// TwinCAT 3 PLC project Modbus
// ProgramVersion: 3.1.4022.7
// libraries:
//   LCLS Vacuum, * (SLAC - LCLS)
//   Tc2_ModbusRTU, * (Beckhoff Automation GmbH)
//   Tc2_ModbusSrv, * (Beckhoff Automation GmbH)
//   Tc2_Standard, * (Beckhoff Automation GmbH)
//   Tc2_System, * (Beckhoff Automation GmbH)
//   Tc3_Module, * (Beckhoff Automation GmbH)
// project tree:
//   / PlcTask.TcTTO
//   POUs/ FB_GaugeModbus.TcPOU, MAIN.TcPOU
//   POUs/Modbus/ p_ModbusRx_OutputCoils.TcPOU, p_ModbusRx_OutputReg.TcPOU, p_ModbusRx_PLCMemory.TcPOU, p_ModbusTx_InputCoils.TcPOU, p_ModbusTx_InputReg.TcPOU, p_ModbusTx_OutputCoils.TcPOU, p_ModbusTx_OutputReg.TcPOU, p_ModbusTx_PLCMemory.TcPOU, p_XLegacyPLCModbus.TcPOU
// real-time tasks:
//   TASK PlcTask: cycle T#10ms, priority 20, ADS port 350

CONFIGURATION Modbus
    RESOURCE PLC ON TwinCAT3
        TASK PlcTask(INTERVAL := T#10ms, PRIORITY := 20);
        PROGRAM MAIN WITH PlcTask : MAIN;
    END_RESOURCE
END_CONFIGURATION

// ---- POUs/MAIN.TcPOU
PROGRAM MAIN
VAR
	test:FB_GaugeModbus;
	
END_VAR

test(IP:='172.21.84.44',nMBAddr:=2048(*8#4000*),iBitOffset:=24);

END_PROGRAM

// ---- POUs/FB_GaugeModbus.TcPOU
FUNCTION_BLOCK FB_GaugeModbus EXTENDS FB_GaugeBase
VAR_INPUT
	IP: STRING;	//IP of Legacy PLC
    nMBAddr	:WORD; //Start address of the Register Memory
	iBitOffset:INT :=24;
	tTimeout :TIME:= T#5s;
END_VAR
VAR_OUTPUT
	VG: ST_VG;
	xNoPLCResponse: BOOL;
END_VAR
VAR
	fbPLCInputCoilsRx	:	FB_MBReadInputs;// (Modbus function 2)
	i_PLC_nBits	:	ARRAY [1..4] OF BYTE;
	ftReset	: F_TRIG; 
	tonRetry : TON;
	ErrCount:INT :=0;
END_VAR

A_ReadMB();

ACTION A_ReadMB:
(*Credit to Alex Wallace*)
(* Modbus Info for Koyo
Modbus Addresses for
Koyo DL05/06/240/250/260/430/440/450 PLCs
PLC Memory Type		| Modbus start address Decimal (octal) | Function codes
Inputs (X)			  2048 (04000)							2
Special Relays (SP)	  3072 (06000)							2
Outputs (Y)			  2048 (04000)							1, 5, 15
Control Relays (C)	  3072 (06000)							1, 5, 15
Timer Contacts (T)	  6144 (014000)							1, 5, 15
Counter Contacts (CT) 6400 (014400)							1, 5, 15
Stage Status Bits (S) 6144 (012000)							1, 5, 15
*)

// Retry after some time
tonRetry.IN := NOT fbPLCInputCoilsRx.bBusy;
tonRetry.PT := T#10S;
tonRetry();

ftReset(CLK:=fbPLCInputCoilsRx.bBusy);
fbPLCInputCoilsRx.bExecute := ftReset.Q OR tonRetry.Q;

fbPLCInputCoilsRx(sIPAddr:=IP, nTCPPort:=502, nQuantity:=24, nMBAddr:=nMBAddr(*+INT_TO_WORD(iBitOffset)*), cbLength:=SIZEOF(i_PLC_nBits),  pDestAddr:=ADR(i_PLC_nBits), tTimeout:=tTimeout);
//if there's a modbus error, set all incoming bits to zero
IF fbPLCInputCoilsRx.bError THEN
	i_PLC_nBits[1].0 := 0;
	i_PLC_nBits[1].1 := 0;
	i_PLC_nBits[1].2 := 0;
	i_PLC_nBits[1].3 := 0;
	i_PLC_nBits[1].4 := 0;
	i_PLC_nBits[1].5 := 0;
	i_PLC_nBits[1].6 := 0;
	i_PLC_nBits[1].7 := 0;
	i_PLC_nBits[2].0 := 0;
	i_PLC_nBits[2].1 := 0;
	i_PLC_nBits[2].2 := 0;
	i_PLC_nBits[2].3 := 0;
	i_PLC_nBits[2].4 := 0;
	i_PLC_nBits[2].5 := 0;
	i_PLC_nBits[2].6 := 0;
	i_PLC_nBits[2].7 := 0;
	VG.xPRESS_OK := FALSE;
	xNoPLCResponse:= TRUE;	
ELSIF NOT ftReset.Q AND fbPLCInputCoilsRx.cbRead > 0 THEN
	xNoPLCResponse:= FALSE;
	VG.rPRESS := 1E-8;
	VG.xPRESS_OK := i_PLC_nBits[0].0;
	fbPLCInputCoilsRx.bExecute :=False;
ELSIF (*ftReset.Q*) NOT (fbPLCInputCoilsRx.bExecute) AND fbPLCInputCoilsRx.cbRead = 0 THEN
	xNoPLCResponse:= TRUE;		
END_IF

// Log Action
tAction(CLK:=   fbPLCInputCoilsRx.bError or xNoPLCResponse);
IF tAction.Q THEN 
ErrCount:= ErrCount+1; 
fbLogger(sMsg:='Modbus read error', eSevr:=TcEventSeverity.Critical);
END_IF
END_ACTION

END_FUNCTION_BLOCK

// ---- POUs/Modbus/p_ModbusRx_OutputCoils.TcPOU
PROGRAM p_ModbusRx_OutputCoils
VAR
END_VAR

//mb_Output_Coils[0];  //System Controls
g_stSystem.xOverrideMode:=mb_Output_Coils[1];  //System Controls
//mb_Output_Coils[2];  //System Controls
//mb_Output_Coils[3];  //System Controls
//mb_Output_Coils[4];  //System Controls
//mb_Output_Coils[5];  //System Controls
//mb_Output_Coils[6];  //System Controls
//mb_Output_Coils[7];  //System Controls
//mb_Output_Coils[8];  //System Controls
//mb_Output_Coils[9];  //System Controls
vgcPBT_VGC_01.xOPN_SW:=mb_Output_Coils[10];  //Valve switch controls
vgcPBT_VGC_02.xOPN_SW:=mb_Output_Coils[11];  //Valve switch controls
vgcPBT_VGC_03.xOPN_SW:=mb_Output_Coils[12];  //Valve switch controls
vgcPBT_VGC_04.xOPN_SW:=mb_Output_Coils[13];  //Valve switch controls
//mb_Output_Coils[14];  //Valve switch controls
//mb_Output_Coils[15];  //Valve switch controls
//mb_Output_Coils[16];  //Valve switch controls
//mb_Output_Coils[17];  //Valve switch controls
//mb_Output_Coils[18];  //Valve switch controls
//mb_Output_Coils[19];  //Valve switch controls
//mb_Output_Coils[20];  //Valve switch controls
//mb_Output_Coils[21];  //Valve switch controls
//mb_Output_Coils[22];  //Valve switch controls
//mb_Output_Coils[23];  //Valve switch controls
//mb_Output_Coils[24];  //Valve switch controls
//mb_Output_Coils[25];  //Valve switch controls
//mb_Output_Coils[26];  //Valve switch controls
//mb_Output_Coils[27];  //Valve switch controls
//mb_Output_Coils[28];  //Valve switch controls
//mb_Output_Coils[29];  //Valve switch controls
//mb_Output_Coils[30];  //Valve switch controls
//mb_Output_Coils[31];  //Valve switch controls
//mb_Output_Coils[32];  //Valve switch controls
//mb_Output_Coils[33];  //Valve switch controls
//mb_Output_Coils[34];  //Valve switch controls
//mb_Output_Coils[35];  //Valve switch controls
//mb_Output_Coils[36];  //Valve switch controls
//mb_Output_Coils[37];  //Valve switch controls
//mb_Output_Coils[38];  //Valve switch controls
//mb_Output_Coils[39];  //Valve switch controls
//mb_Output_Coils[40];  //Valve switch controls
//mb_Output_Coils[41];  //Valve switch controls
//mb_Output_Coils[42];  //Valve switch controls
//mb_Output_Coils[43];  //Valve switch controls
//mb_Output_Coils[44];  //Valve switch controls
//mb_Output_Coils[45];  //Valve switch controls
//mb_Output_Coils[46];  //Valve switch controls
//mb_Output_Coils[47];  //Valve switch controls
//mb_Output_Coils[48];  //Valve switch controls
//mb_Output_Coils[49];  //Valve switch controls
//mb_Output_Coils[50];  //Valve switch controls
//mb_Output_Coils[51];  //Valve switch controls
//mb_Output_Coils[52];  //Valve switch controls
//mb_Output_Coils[53];  //Valve switch controls
//mb_Output_Coils[54];  //Valve switch controls
//mb_Output_Coils[55];  //Valve switch controls
//mb_Output_Coils[56];  //Valve switch controls
//mb_Output_Coils[57];  //Valve switch controls
//mb_Output_Coils[58];  //Valve switch controls
//mb_Output_Coils[59];  //Valve switch controls
//mb_Output_Coils[60];  //Valve switch controls
//mb_Output_Coils[61];  //Valve switch controls
//mb_Output_Coils[62];  //Valve switch controls
//mb_Output_Coils[63];  //Valve switch controls
//mb_Output_Coils[64];  //Valve switch controls
//mb_Output_Coils[65];  //Valve switch controls
//mb_Output_Coils[66];  //Valve switch controls
//mb_Output_Coils[67];  //Valve switch controls
//mb_Output_Coils[68];  //Valve switch controls
//mb_Output_Coils[69];  //Valve switch controls
//mb_Output_Coils[70];  //Turbo Controls
//mb_Output_Coils[71];  //Turbo Controls
//mb_Output_Coils[72];  //Turbo Controls
//mb_Output_Coils[74];  //Turbo Controls
//mb_Output_Coils[75];  //Turbo Controls
//mb_Output_Coils[76];  //Turbo Controls
//mb_Output_Coils[77];  //Turbo Controls
//mb_Output_Coils[78];  //Turbo Controls
//mb_Output_Coils[79];  //Turbo Controls
//mb_Output_Coils[80];  //Turbo Controls
//mb_Output_Coils[81];  //Turbo Controls
//mb_Output_Coils[82];  //Turbo Controls
//mb_Output_Coils[83];  //Turbo Controls
//mb_Output_Coils[84];  //Turbo Controls
//mb_Output_Coils[85];  //Turbo Controls
//mb_Output_Coils[86];  //Turbo Controls
//mb_Output_Coils[87];  //Turbo Controls
//mb_Output_Coils[88];  //Turbo Controls
//mb_Output_Coils[89];  //Turbo Controls
//mb_Output_Coils[90];  //Turbo Controls
//mb_Output_Coils[91];  //Turbo Controls
//mb_Output_Coils[92];  //Turbo Controls
//mb_Output_Coils[93];  //Turbo Controls
//mb_Output_Coils[94];  //Turbo Controls
//mb_Output_Coils[95];  //Turbo Controls
//mb_Output_Coils[96];  //Turbo Controls
//mb_Output_Coils[97];  //Turbo Controls
//mb_Output_Coils[98];  //Turbo Controls
//mb_Output_Coils[99];  //Turbo Controls
//mb_Output_Coils[100];  //Turbo Controls
//mb_Output_Coils[101];  //Turbo Controls
//mb_Output_Coils[102];  //Turbo Controls
//mb_Output_Coils[103];  //Turbo Controls
//mb_Output_Coils[104];  //Turbo Controls
//mb_Output_Coils[105];  //Turbo Controls
//mb_Output_Coils[106];  //Turbo Controls
//mb_Output_Coils[107];  //Turbo Controls
//mb_Output_Coils[108];  //Turbo Controls
//mb_Output_Coils[109];  //Turbo Controls
//mb_Output_Coils[110];  //Turbo Controls
//mb_Output_Coils[111];  //Turbo Controls
//mb_Output_Coils[112];  //Turbo Controls
//mb_Output_Coils[113];  //Turbo Controls
//mb_Output_Coils[114];  //Turbo Controls
//mb_Output_Coils[115];  //Turbo Controls
//mb_Output_Coils[116];  //Turbo Controls
//mb_Output_Coils[117];  //Turbo Controls
//mb_Output_Coils[118];  //Turbo Controls
//mb_Output_Coils[119];  //Turbo Controls
vgPBT_GCC_02.xHV_SW:=mb_Output_Coils[120];  //CC HV Enable
vgPBT_GCC_04.xHV_SW:=mb_Output_Coils[121];  //CC HV Enable
vgPBT_GCC_06.xHV_SW:=mb_Output_Coils[122];  //CC HV Enable
vgPBT_GCC_07.xHV_SW:=mb_Output_Coils[123];  //CC HV Enable
vgPBT_GCC_09.xHV_SW:=mb_Output_Coils[124];  //CC HV Enable
//mb_Output_Coils[125];  //CC HV Enable
//mb_Output_Coils[126];  //CC HV Enable
//mb_Output_Coils[127];  //CC HV Enable
//mb_Output_Coils[128];  //CC HV Enable
//mb_Output_Coils[129];  //CC HV Enable
//mb_Output_Coils[130];  //CC HV Enable
//mb_Output_Coils[131];  //CC HV Enable
//mb_Output_Coils[132];  //CC HV Enable
//mb_Output_Coils[133];  //CC HV Enable
//mb_Output_Coils[134];  //CC HV Enable
//mb_Output_Coils[135];  //CC HV Enable
//mb_Output_Coils[136];  //CC HV Enable
//mb_Output_Coils[137];  //CC HV Enable
//mb_Output_Coils[138];  //CC HV Enable
//mb_Output_Coils[139];  //CC HV Enable
//mb_Output_Coils[140];  //CC HV Enable
//mb_Output_Coils[141];  //CC HV Enable
//mb_Output_Coils[142];  //CC HV Enable
//mb_Output_Coils[143];  //CC HV Enable
//mb_Output_Coils[144];  //CC HV Enable
//mb_Output_Coils[145];  //CC HV Enable
//mb_Output_Coils[146];  //CC HV Enable
//mb_Output_Coils[147];  //CC HV Enable
//mb_Output_Coils[148];  //CC HV Enable
//mb_Output_Coils[149];  //CC HV Enable
//mb_Output_Coils[150];  //CC HV Enable
//mb_Output_Coils[151];  //CC HV Enable
//mb_Output_Coils[152];  //CC HV Enable
//mb_Output_Coils[153];  //CC HV Enable
//mb_Output_Coils[154];  //CC HV Enable
//mb_Output_Coils[155];  //CC HV Enable
//mb_Output_Coils[156];  //CC HV Enable
//mb_Output_Coils[157];  //CC HV Enable
//mb_Output_Coils[158];  //CC HV Enable
//mb_Output_Coils[159];  //CC HV Enable
//mb_Output_Coils[160];  //
//mb_Output_Coils[161];  //
//mb_Output_Coils[162];  //
//mb_Output_Coils[163];  //
//mb_Output_Coils[164];  //
//mb_Output_Coils[165];  //
//mb_Output_Coils[166];  //
//mb_Output_Coils[167];  //
//mb_Output_Coils[168];  //
//mb_Output_Coils[169];  //
//mb_Output_Coils[170];  //
//mb_Output_Coils[171];  //
//mb_Output_Coils[172];  //
//mb_Output_Coils[173];  //
//mb_Output_Coils[174];  //
//mb_Output_Coils[175];  //
//mb_Output_Coils[176];  //
//mb_Output_Coils[177];  //
//mb_Output_Coils[178];  //
//mb_Output_Coils[179];  //
//mb_Output_Coils[180];  //
//mb_Output_Coils[181];  //
//mb_Output_Coils[182];  //
//mb_Output_Coils[183];  //
//mb_Output_Coils[184];  //
//mb_Output_Coils[185];  //
//mb_Output_Coils[186];  //
//mb_Output_Coils[187];  //
//mb_Output_Coils[188];  //
//mb_Output_Coils[189];  //
//mb_Output_Coils[190];  //
//mb_Output_Coils[191];  //
//mb_Output_Coils[192];  //
//mb_Output_Coils[193];  //
//mb_Output_Coils[194];  //
//mb_Output_Coils[195];  //
//mb_Output_Coils[196];  //
//mb_Output_Coils[197];  //
//mb_Output_Coils[198];  //
//mb_Output_Coils[199];  //
vgcPBT_VGC_01.xOvrdOpn:=mb_Output_Coils[200];  //Valve overrides
vgcPBT_VGC_02.xOvrdOpn:=mb_Output_Coils[201];  //Valve overrides
vgcPBT_VGC_03.xOvrdOpn:=mb_Output_Coils[202];  //Valve overrides
vgcPBT_VGC_04.xOvrdOpn:=mb_Output_Coils[203];  //Valve overrides
//mb_Output_Coils[204];  //
//mb_Output_Coils[205];  //
//mb_Output_Coils[206];  //
//mb_Output_Coils[207];  //
//mb_Output_Coils[208];  //
//mb_Output_Coils[209];  //
//mb_Output_Coils[210];  //
//mb_Output_Coils[211];  //
//mb_Output_Coils[212];  //
//mb_Output_Coils[213];  //
//mb_Output_Coils[214];  //
//mb_Output_Coils[215];  //
//mb_Output_Coils[216];  //
//mb_Output_Coils[217];  //
//mb_Output_Coils[218];  //
//mb_Output_Coils[219];  //
//mb_Output_Coils[220];  //
//mb_Output_Coils[221];  //
//mb_Output_Coils[222];  //
//mb_Output_Coils[223];  //
//mb_Output_Coils[224];  //
//mb_Output_Coils[225];  //
//mb_Output_Coils[226];  //
//mb_Output_Coils[227];  //
//mb_Output_Coils[228];  //
//mb_Output_Coils[229];  //
//mb_Output_Coils[230];  //
//mb_Output_Coils[231];  //
//mb_Output_Coils[232];  //
//mb_Output_Coils[233];  //
//mb_Output_Coils[234];  //
//mb_Output_Coils[235];  //
//mb_Output_Coils[236];  //
//mb_Output_Coils[237];  //
//mb_Output_Coils[238];  //
//mb_Output_Coils[239];  //
//mb_Output_Coils[240];  //
//mb_Output_Coils[241];  //
//mb_Output_Coils[242];  //
//mb_Output_Coils[243];  //
//mb_Output_Coils[244];  //
//mb_Output_Coils[245];  //
//mb_Output_Coils[246];  //
//mb_Output_Coils[247];  //
//mb_Output_Coils[248];  //
//mb_Output_Coils[249];  //
//mb_Output_Coils[250];  //
//mb_Output_Coils[251];  //
//mb_Output_Coils[252];  //
//mb_Output_Coils[253];  //
//mb_Output_Coils[254];  //
//mb_Output_Coils[255];  //

END_PROGRAM

// ---- POUs/Modbus/p_ModbusRx_OutputReg.TcPOU
PROGRAM p_ModbusRx_OutputReg
VAR
END_VAR

//mb_Output_Registers[0];  //System parameters
//mb_Output_Registers[1];  //System parameters
//mb_Output_Registers[2];  //System parameters
//mb_Output_Registers[3];  //System parameters
//mb_Output_Registers[4];  //System parameters
//mb_Output_Registers[5];  //System parameters
//mb_Output_Registers[6];  //System parameters
//mb_Output_Registers[7];  //System parameters
//mb_Output_Registers[8];  //System parameters
//mb_Output_Registers[9];  //System parameters
//mb_Output_Registers[10];  //VG setpoint
//mb_Output_Registers[11];  //VG setpoint
//mb_Output_Registers[12];  //VG setpoint
//mb_Output_Registers[13];  //VG setpoint
//mb_Output_Registers[14];  //VG setpoint
//mb_Output_Registers[15];  //VG setpoint
//mb_Output_Registers[16];  //VG setpoint
//mb_Output_Registers[17];  //VG setpoint
//mb_Output_Registers[18];  //VG setpoint
//mb_Output_Registers[19];  //VG setpoint
//mb_Output_Registers[20];  //VG setpoint
//mb_Output_Registers[21];  //VG setpoint
//mb_Output_Registers[22];  //VG setpoint
//mb_Output_Registers[23];  //VG setpoint
//mb_Output_Registers[24];  //VG setpoint
//mb_Output_Registers[25];  //VG setpoint
//mb_Output_Registers[26];  //VG setpoint
//mb_Output_Registers[27];  //VG setpoint
//mb_Output_Registers[28];  //VG setpoint
//mb_Output_Registers[29];  //VG setpoint
//mb_Output_Registers[30];  //VG setpoint
//mb_Output_Registers[31];  //VG setpoint
//mb_Output_Registers[32];  //VG setpoint
//mb_Output_Registers[33];  //VG setpoint
//mb_Output_Registers[34];  //VG setpoint
//mb_Output_Registers[35];  //VG setpoint
//mb_Output_Registers[36];  //VG setpoint
//mb_Output_Registers[37];  //VG setpoint
//mb_Output_Registers[38];  //VG setpoint
//mb_Output_Registers[39];  //VG setpoint
//mb_Output_Registers[40];  //VG setpoint
//mb_Output_Registers[41];  //VG setpoint
//mb_Output_Registers[42];  //VG setpoint
//mb_Output_Registers[43];  //VG setpoint
//mb_Output_Registers[44];  //VG setpoint
//mb_Output_Registers[45];  //VG setpoint
//mb_Output_Registers[46];  //VG setpoint
//mb_Output_Registers[47];  //VG setpoint
//mb_Output_Registers[48];  //VG setpoint
//mb_Output_Registers[49];  //VG setpoint
//mb_Output_Registers[50];  //VG setpoint
//mb_Output_Registers[51];  //VG setpoint
//mb_Output_Registers[52];  //VG setpoint
//mb_Output_Registers[53];  //VG setpoint
//mb_Output_Registers[54];  //VG setpoint
//mb_Output_Registers[55];  //VG setpoint
//mb_Output_Registers[56];  //VG setpoint
//mb_Output_Registers[57];  //VG setpoint
//mb_Output_Registers[58];  //VG setpoint
//mb_Output_Registers[59];  //VG setpoint
//mb_Output_Registers[60];  //default
//mb_Output_Registers[61];  //default
//mb_Output_Registers[62];  //default
//mb_Output_Registers[63];  //default
//mb_Output_Registers[64];  //default
//mb_Output_Registers[65];  //default
//mb_Output_Registers[66];  //default
//mb_Output_Registers[67];  //default
//mb_Output_Registers[68];  //default
//mb_Output_Registers[69];  //default
//mb_Output_Registers[70];  //default
//mb_Output_Registers[71];  //default
//mb_Output_Registers[72];  //default
//mb_Output_Registers[73];  //default
//mb_Output_Registers[74];  //default
//mb_Output_Registers[75];  //default
//mb_Output_Registers[76];  //default
//mb_Output_Registers[77];  //default
//mb_Output_Registers[78];  //default
//mb_Output_Registers[79];  //default
//mb_Output_Registers[80];  //default
//mb_Output_Registers[81];  //default
//mb_Output_Registers[82];  //default
//mb_Output_Registers[83];  //default
//mb_Output_Registers[84];  //default
//mb_Output_Registers[85];  //default
//mb_Output_Registers[86];  //default
//mb_Output_Registers[87];  //default
//mb_Output_Registers[88];  //default
//mb_Output_Registers[89];  //default
//mb_Output_Registers[90];  //default
//mb_Output_Registers[91];  //default
//mb_Output_Registers[92];  //default
//mb_Output_Registers[93];  //default
//mb_Output_Registers[94];  //default
//mb_Output_Registers[95];  //default
//mb_Output_Registers[96];  //default
//mb_Output_Registers[97];  //default
//mb_Output_Registers[98];  //default
//mb_Output_Registers[99];  //default
//mb_Output_Registers[100];  //default
//mb_Output_Registers[101];  //default
//mb_Output_Registers[102];  //default
//mb_Output_Registers[103];  //default
//mb_Output_Registers[104];  //default
//mb_Output_Registers[105];  //default
//mb_Output_Registers[106];  //default
//mb_Output_Registers[107];  //default
//mb_Output_Registers[108];  //default
//mb_Output_Registers[109];  //default
//mb_Output_Registers[110];  //default
//mb_Output_Registers[111];  //default
//mb_Output_Registers[112];  //default
//mb_Output_Registers[113];  //default
//mb_Output_Registers[114];  //default
//mb_Output_Registers[115];  //default
//mb_Output_Registers[116];  //default
//mb_Output_Registers[117];  //default
//mb_Output_Registers[118];  //default
//mb_Output_Registers[119];  //default
//mb_Output_Registers[120];  //default
//mb_Output_Registers[121];  //default
//mb_Output_Registers[122];  //default
//mb_Output_Registers[123];  //default
//mb_Output_Registers[124];  //default
//mb_Output_Registers[125];  //default
//mb_Output_Registers[126];  //default
//mb_Output_Registers[127];  //default
//mb_Output_Registers[128];  //default
//mb_Output_Registers[129];  //default
//mb_Output_Registers[130];  //default
//mb_Output_Registers[131];  //default
//mb_Output_Registers[132];  //default
//mb_Output_Registers[133];  //default
//mb_Output_Registers[134];  //default
//mb_Output_Registers[135];  //default
//mb_Output_Registers[136];  //default
//mb_Output_Registers[137];  //default
//mb_Output_Registers[138];  //default
//mb_Output_Registers[139];  //default
//mb_Output_Registers[140];  //default
//mb_Output_Registers[141];  //default
//mb_Output_Registers[142];  //default
//mb_Output_Registers[143];  //default
//mb_Output_Registers[144];  //default
//mb_Output_Registers[145];  //default
//mb_Output_Registers[146];  //default
//mb_Output_Registers[147];  //default
//mb_Output_Registers[148];  //default
//mb_Output_Registers[149];  //default
//mb_Output_Registers[150];  //default
//mb_Output_Registers[151];  //default
//mb_Output_Registers[152];  //default
//mb_Output_Registers[153];  //default
//mb_Output_Registers[154];  //default
//mb_Output_Registers[155];  //default
//mb_Output_Registers[156];  //default
//mb_Output_Registers[157];  //default
//mb_Output_Registers[158];  //default
//mb_Output_Registers[159];  //default
//mb_Output_Registers[160];  //default
//mb_Output_Registers[161];  //default
//mb_Output_Registers[162];  //default
//mb_Output_Registers[163];  //default
//mb_Output_Registers[164];  //default
//mb_Output_Registers[165];  //default
//mb_Output_Registers[166];  //default
//mb_Output_Registers[167];  //default
//mb_Output_Registers[168];  //default
//mb_Output_Registers[169];  //default
//mb_Output_Registers[170];  //default
//mb_Output_Registers[171];  //default
//mb_Output_Registers[172];  //default
//mb_Output_Registers[173];  //default
//mb_Output_Registers[174];  //default
//mb_Output_Registers[175];  //default
//mb_Output_Registers[176];  //default
//mb_Output_Registers[177];  //default
//mb_Output_Registers[178];  //default
//mb_Output_Registers[179];  //default
//mb_Output_Registers[180];  //default
//mb_Output_Registers[181];  //default
//mb_Output_Registers[182];  //default
//mb_Output_Registers[183];  //default
//mb_Output_Registers[184];  //default
//mb_Output_Registers[185];  //default
//mb_Output_Registers[186];  //default
//mb_Output_Registers[187];  //default
//mb_Output_Registers[188];  //default
//mb_Output_Registers[189];  //default
//mb_Output_Registers[190];  //default
//mb_Output_Registers[191];  //default
//mb_Output_Registers[192];  //default
//mb_Output_Registers[193];  //default
//mb_Output_Registers[194];  //default
//mb_Output_Registers[195];  //default
//mb_Output_Registers[196];  //default
//mb_Output_Registers[197];  //default
//mb_Output_Registers[198];  //default
//mb_Output_Registers[199];  //default
//mb_Output_Registers[200];  //default
//mb_Output_Registers[201];  //default
//mb_Output_Registers[202];  //default
//mb_Output_Registers[203];  //default
//mb_Output_Registers[204];  //default
//mb_Output_Registers[205];  //default
//mb_Output_Registers[206];  //default
//mb_Output_Registers[207];  //default
//mb_Output_Registers[208];  //default
//mb_Output_Registers[209];  //default
//mb_Output_Registers[210];  //default
//mb_Output_Registers[211];  //default
//mb_Output_Registers[212];  //default
//mb_Output_Registers[213];  //default
//mb_Output_Registers[214];  //default
//mb_Output_Registers[215];  //default
//mb_Output_Registers[216];  //default
//mb_Output_Registers[217];  //default
//mb_Output_Registers[218];  //default
//mb_Output_Registers[219];  //default
//mb_Output_Registers[220];  //default
//mb_Output_Registers[221];  //default
//mb_Output_Registers[222];  //default
//mb_Output_Registers[223];  //default
//mb_Output_Registers[224];  //default
//mb_Output_Registers[225];  //default
//mb_Output_Registers[226];  //default
//mb_Output_Registers[227];  //default
//mb_Output_Registers[228];  //default
//mb_Output_Registers[229];  //default
//mb_Output_Registers[230];  //default
//mb_Output_Registers[231];  //default
//mb_Output_Registers[232];  //default
//mb_Output_Registers[233];  //default
//mb_Output_Registers[234];  //default
//mb_Output_Registers[235];  //default
//mb_Output_Registers[236];  //default
//mb_Output_Registers[237];  //default
//mb_Output_Registers[238];  //default
//mb_Output_Registers[239];  //default
//mb_Output_Registers[240];  //default
//mb_Output_Registers[241];  //default
//mb_Output_Registers[242];  //default
//mb_Output_Registers[243];  //default
//mb_Output_Registers[244];  //default
//mb_Output_Registers[245];  //default
//mb_Output_Registers[246];  //default
//mb_Output_Registers[247];  //default
//mb_Output_Registers[248];  //default
//mb_Output_Registers[249];  //default
//mb_Output_Registers[250];  //default
//mb_Output_Registers[251];  //default
//mb_Output_Registers[252];  //default
//mb_Output_Registers[253];  //default
//mb_Output_Registers[254];  //default
//mb_Output_Registers[255];  //default

END_PROGRAM

// ---- POUs/Modbus/p_ModbusRx_PLCMemory.TcPOU
PROGRAM p_ModbusRx_PLCMemory
VAR
END_VAR

MEMCPY(destAddr:=ADR(mb_PLC_Memory[70]), srcAddr:=ADR(vgPBT_GCC_02.rVAC_SP), n:=SIZEOF(vgPBT_GCC_02.rVAC_SP));  //VG pressure sp readbacks
MEMCPY(destAddr:=ADR(mb_PLC_Memory[72]), srcAddr:=ADR(vgPBT_GPI_02.rVAC_SP), n:=SIZEOF(vgPBT_GPI_02.rVAC_SP));  //VG pressure sp readbacks

MEMCPY(destAddr:=ADR(mb_PLC_Memory[74]), srcAddr:=ADR(vgPBT_GCC_04.rVAC_SP), n:=SIZEOF(vgPBT_GCC_04.rVAC_SP));  //VG pressure sp readbacks
MEMCPY(destAddr:=ADR(mb_PLC_Memory[76]), srcAddr:=ADR(vgPBT_GPI_04.rVAC_SP), n:=SIZEOF(vgPBT_GPI_04.rVAC_SP));  //VG pressure sp readbacks

MEMCPY(destAddr:=ADR(mb_PLC_Memory[78]), srcAddr:=ADR(vgPBT_GCC_06.rVAC_SP), n:=SIZEOF(vgPBT_GCC_06.rVAC_SP));  //VG pressure sp readbacks
MEMCPY(destAddr:=ADR(mb_PLC_Memory[80]), srcAddr:=ADR(vgPBT_GPI_06.rVAC_SP), n:=SIZEOF(vgPBT_GPI_06.rVAC_SP));  //VG pressure sp readbacks

MEMCPY(destAddr:=ADR(mb_PLC_Memory[82]), srcAddr:=ADR(vgPBT_GCC_07.rVAC_SP), n:=SIZEOF(vgPBT_GCC_07.rVAC_SP));  //VG pressure sp readbacks
MEMCPY(destAddr:=ADR(mb_PLC_Memory[84]), srcAddr:=ADR(vgPBT_GPI_07.rVAC_SP), n:=SIZEOF(vgPBT_GPI_07.rVAC_SP));  //VG pressure sp readbacks

MEMCPY(destAddr:=ADR(mb_PLC_Memory[86]), srcAddr:=ADR(vgPBT_GCC_09.rVAC_SP), n:=SIZEOF(vgPBT_GCC_09.rVAC_SP));  //VG pressure sp readbacks
MEMCPY(destAddr:=ADR(mb_PLC_Memory[88]), srcAddr:=ADR(vgPBT_GPI_09.rVAC_SP), n:=SIZEOF(vgPBT_GPI_09.rVAC_SP));  //VG pressure sp readbacks

END_PROGRAM

// ---- POUs/Modbus/p_ModbusTx_InputCoils.TcPOU
PROGRAM p_ModbusTx_InputCoils
VAR
	
END_VAR

VAR_OUTPUT
	

	XHV_DIS: BOOL;
END_VAR

mb_Input_Coils[0]:=FALSE;  //default
//mb_Input_Coils[1]:=i_xMFX_ppsStopperPos_Out;  //default
//mb_Input_Coils[2]:=i_xMFX_ppsStopperPos_In;  //default
mb_Input_Coils[3]:=q_xXCS_MPSOK;  //default
mb_Input_Coils[4]:=g_xIOState;  //default
//mb_Input_Coils[5]:=i_xDG1_MMS01_OUT;  //default
mb_Input_Coils[6]:=FALSE;  //default
mb_Input_Coils[7]:=FALSE;  //default
mb_Input_Coils[8]:=FALSE;  //default
mb_Input_Coils[9]:=FALSE;  //default
mb_Input_Coils[10]:=vgcPBT_VGC_01.i_xOpnLS;  //Valve position readbacks
mb_Input_Coils[11]:=vgcPBT_VGC_01.i_xClsLS;  //Valve position readbacks
mb_Input_Coils[12]:=vgcPBT_VGC_02.i_xOpnLS;  //Valve position readbacks
mb_Input_Coils[13]:=vgcPBT_VGC_02.i_xClsLS;  //Valve position readbacks
mb_Input_Coils[14]:=vgcPBT_VGC_03.i_xOpnLS;  //Valve position readbacks
mb_Input_Coils[15]:=vgcPBT_VGC_03.i_xClsLS;  //Valve position readbacks
mb_Input_Coils[16]:=vgcPBT_VGC_04.i_xOpnLS;  //Valve position readbacks
mb_Input_Coils[17]:=vgcPBT_VGC_04.i_xClsLS;  //Valve position readbacks
mb_Input_Coils[18]:=FALSE;  //Valve position readbacks
mb_Input_Coils[19]:=FALSE;  //Valve position readbacks
mb_Input_Coils[20]:=FALSE; //Valve position readbacks
mb_Input_Coils[21]:=FALSE;  //Valve position readbacks
mb_Input_Coils[22]:=FALSE;  //Valve position readbacks
mb_Input_Coils[23]:=FALSE;  //Valve position readbacks
mb_Input_Coils[24]:=FALSE;  //Valve position readbacks
mb_Input_Coils[25]:=FALSE;  //Valve position readbacks
mb_Input_Coils[26]:=FALSE;  //Valve position readbacks
mb_Input_Coils[27]:=FALSE;  //Valve position readbacks
mb_Input_Coils[28]:=FALSE;  //Valve position readbacks
mb_Input_Coils[29]:=FALSE;  //Valve position readbacks
mb_Input_Coils[30]:=FALSE;  //Valve position readbacks
mb_Input_Coils[31]:=FALSE;  //Valve position readbacks
mb_Input_Coils[32]:=FALSE;  //Valve position readbacks
mb_Input_Coils[33]:=FALSE;  //Valve position readbacks
mb_Input_Coils[34]:=FALSE;  //Valve position readbacks
mb_Input_Coils[35]:=FALSE;  //Valve position readbacks
mb_Input_Coils[36]:=FALSE;  //Valve position readbacks
mb_Input_Coils[37]:=FALSE;  //Valve position readbacks
mb_Input_Coils[38]:=FALSE;  //Valve position readbacks
mb_Input_Coils[39]:=FALSE;  //Valve position readbacks
mb_Input_Coils[40]:=FALSE;  //Valve position readbacks
mb_Input_Coils[41]:=FALSE;  //Valve position readbacks
mb_Input_Coils[42]:=FALSE;  //Valve position readbacks
mb_Input_Coils[43]:=FALSE;  //Valve position readbacks
mb_Input_Coils[44]:=FALSE;  //Valve position readbacks
mb_Input_Coils[45]:=FALSE;  //Valve position readbacks
mb_Input_Coils[46]:=FALSE;  //Valve position readbacks
mb_Input_Coils[47]:=FALSE;  //Valve position readbacks
mb_Input_Coils[48]:=FALSE;  //Valve position readbacks
mb_Input_Coils[49]:=FALSE;  //Valve position readbacks
mb_Input_Coils[50]:=FALSE;  //Valve position readbacks
mb_Input_Coils[51]:=FALSE;  //Valve position readbacks
mb_Input_Coils[52]:=FALSE;  //Valve position readbacks
mb_Input_Coils[53]:=FALSE;  //Valve position readbacks
mb_Input_Coils[54]:=FALSE;  //Valve position readbacks
mb_Input_Coils[55]:=FALSE;  //Valve position readbacks
mb_Input_Coils[56]:=FALSE;  //Valve position readbacks
mb_Input_Coils[57]:=FALSE;  //Valve position readbacks
mb_Input_Coils[58]:=FALSE;  //Valve position readbacks
mb_Input_Coils[59]:=FALSE;  //Valve position readbacks
mb_Input_Coils[60]:=vgcPBT_VGC_01.xOPN_OK;  //Valve position readbacks
mb_Input_Coils[61]:=vgcPBT_VGC_02.xOPN_OK;  //Valve position readbacks
mb_Input_Coils[62]:=vgcPBT_VGC_03.xOPN_OK;  //Valve position readbacks
mb_Input_Coils[63]:=vgcPBT_VGC_04.xOPN_OK;  //Valve position readbacks
mb_Input_Coils[64]:=FALSE;  //Valve position readbacks
mb_Input_Coils[65]:=FALSE;  //Valve position readbacks
mb_Input_Coils[66]:=FALSE;  //Valve position readbacks
mb_Input_Coils[67]:=FALSE;  //Valve position readbacks
mb_Input_Coils[68]:=FALSE;  //Valve position readbacks
mb_Input_Coils[69]:=FALSE;  //Valve position readbacks
mb_Input_Coils[70]:=FALSE;  //Valve position readbacks
mb_Input_Coils[71]:=FALSE;  //Valve position readbacks
mb_Input_Coils[72]:=FALSE;  //Valve position readbacks
mb_Input_Coils[73]:=FALSE;  //Valve position readbacks
mb_Input_Coils[74]:=FALSE;  //Valve position readbacks
mb_Input_Coils[75]:=FALSE;  //Valve position readbacks
mb_Input_Coils[76]:=FALSE;  //Valve position readbacks
mb_Input_Coils[77]:=FALSE;  //Valve position readbacks
mb_Input_Coils[78]:=FALSE;  //Valve position readbacks
mb_Input_Coils[79]:=FALSE;  //Valve position readbacks
mb_Input_Coils[80]:=FALSE;  //Valve position readbacks
mb_Input_Coils[81]:=FALSE;  //Valve position readbacks
mb_Input_Coils[82]:=FALSE;  //Valve position readbacks
mb_Input_Coils[83]:=FALSE;  //Valve position readbacks
mb_Input_Coils[84]:=FALSE;  //Valve position readbacks
mb_Input_Coils[85]:=FALSE;  //Valve position readbacks
mb_Input_Coils[86]:=FALSE;  //Valve position readbacks
mb_Input_Coils[87]:=FALSE;  //Valve position readbacks
mb_Input_Coils[88]:=FALSE;  //Valve position readbacks
mb_Input_Coils[89]:=FALSE;  //Valve position readbacks
mb_Input_Coils[90]:=FALSE;  //Valve position readbacks
mb_Input_Coils[91]:=FALSE;  //Valve position readbacks
mb_Input_Coils[92]:=FALSE;  //Valve position readbacks
mb_Input_Coils[93]:=FALSE;  //Valve position readbacks
mb_Input_Coils[94]:=FALSE;  //Valve position readbacks
mb_Input_Coils[95]:=FALSE;  //Valve position readbacks
mb_Input_Coils[96]:=FALSE;  //Valve position readbacks
mb_Input_Coils[97]:=FALSE;  //Valve position readbacks
mb_Input_Coils[98]:=FALSE;  //Valve position readbacks
mb_Input_Coils[99]:=FALSE;  //Valve position readbacks
mb_Input_Coils[100]:=FALSE;  //Valve position readbacks
mb_Input_Coils[101]:=FALSE;  //Valve position readbacks
mb_Input_Coils[102]:=FALSE;  //Valve position readbacks
mb_Input_Coils[103]:=FALSE;  //Valve position readbacks
mb_Input_Coils[104]:=FALSE;  //Valve position readbacks
mb_Input_Coils[105]:=FALSE;  //Valve position readbacks
mb_Input_Coils[106]:=FALSE;  //Valve position readbacks
mb_Input_Coils[107]:=FALSE;  //Valve position readbacks
mb_Input_Coils[108]:=FALSE;  //Valve position readbacks
mb_Input_Coils[109]:=FALSE;  //Valve position readbacks
mb_Input_Coils[110]:=FALSE;  //Valve position readbacks
mb_Input_Coils[111]:=FALSE;  //Valve position readbacks
mb_Input_Coils[112]:=FALSE;  //Valve position readbacks
mb_Input_Coils[113]:=FALSE;  //Valve position readbacks
mb_Input_Coils[114]:=FALSE;  //Valve position readbacks
mb_Input_Coils[115]:=FALSE;  //Valve position readbacks
mb_Input_Coils[116]:=FALSE;  //Valve position readbacks
mb_Input_Coils[117]:=FALSE;  //Valve position readbacks
mb_Input_Coils[118]:=FALSE;  //Valve position readbacks
mb_Input_Coils[119]:=FALSE;  //Valve position readbacks
mb_Input_Coils[120]:=FALSE;  //Turbo pump readbacks
mb_Input_Coils[121]:=FALSE;  //Turbo pump readbacks
mb_Input_Coils[122]:=FALSE;  //Turbo pump readbacks
mb_Input_Coils[123]:=FALSE;  //Turbo pump readbacks
mb_Input_Coils[124]:=FALSE;  //Turbo pump readbacks
mb_Input_Coils[125]:=FALSE;  //Turbo pump readbacks
mb_Input_Coils[126]:=FALSE;  //Turbo pump readbacks
mb_Input_Coils[127]:=FALSE;  //Turbo pump readbacks
mb_Input_Coils[128]:=FALSE;  //Turbo pump readbacks
mb_Input_Coils[129]:=FALSE;  //Turbo pump readbacks
mb_Input_Coils[130]:=FALSE;  //Turbo pump readbacks
mb_Input_Coils[131]:=FALSE;  //Turbo pump readbacks
mb_Input_Coils[132]:=FALSE;  //Turbo pump readbacks
mb_Input_Coils[133]:=FALSE;  //Turbo pump readbacks
mb_Input_Coils[134]:=FALSE;  //Turbo pump readbacks
mb_Input_Coils[135]:=FALSE;  //Turbo pump readbacks
mb_Input_Coils[136]:=FALSE;  //Turbo pump readbacks
mb_Input_Coils[137]:=FALSE;  //Turbo pump readbacks
mb_Input_Coils[138]:=FALSE;  //Turbo pump readbacks
mb_Input_Coils[139]:=FALSE;  //Turbo pump readbacks
mb_Input_Coils[140]:=FALSE;  //Turbo pump readbacks
mb_Input_Coils[141]:=FALSE;  //Turbo pump readbacks
mb_Input_Coils[142]:=FALSE;  //Turbo pump readbacks
mb_Input_Coils[143]:=FALSE;  //Turbo pump readbacks
mb_Input_Coils[144]:=FALSE;  //Turbo pump readbacks
mb_Input_Coils[145]:=FALSE;  //Turbo pump readbacks
mb_Input_Coils[146]:=FALSE;  //Turbo pump readbacks
mb_Input_Coils[147]:=FALSE;  //Turbo pump readbacks
mb_Input_Coils[148]:=FALSE;  //Turbo pump readbacks
mb_Input_Coils[149]:=FALSE;  //Turbo pump readbacks
mb_Input_Coils[150]:=FALSE;  //Turbo pump readbacks
mb_Input_Coils[151]:=FALSE;  //Turbo pump readbacks
mb_Input_Coils[152]:=FALSE;  //Turbo pump readbacks
mb_Input_Coils[153]:=FALSE;  //Turbo pump readbacks
mb_Input_Coils[154]:=FALSE;  //Turbo pump readbacks
mb_Input_Coils[155]:=FALSE;  //Turbo pump readbacks
mb_Input_Coils[156]:=FALSE;  //Turbo pump readbacks
mb_Input_Coils[157]:=FALSE;  //Turbo pump readbacks
mb_Input_Coils[158]:=FALSE;  //Turbo pump readbacks
mb_Input_Coils[159]:=FALSE;  //Turbo pump readbacks
mb_Input_Coils[160]:=FALSE;  //Turbo pump readbacks
mb_Input_Coils[161]:=FALSE;  //Turbo pump readbacks
mb_Input_Coils[162]:=FALSE;  //Turbo pump readbacks
mb_Input_Coils[163]:=FALSE;  //Turbo pump readbacks
mb_Input_Coils[164]:=FALSE;  //Turbo pump readbacks
mb_Input_Coils[165]:=FALSE;  //Turbo pump readbacks
mb_Input_Coils[166]:=FALSE;  //Turbo pump readbacks
mb_Input_Coils[167]:=FALSE;  //Turbo pump readbacks
mb_Input_Coils[168]:=FALSE;  //Turbo pump readbacks
mb_Input_Coils[169]:=FALSE;  //Turbo pump readbacks
mb_Input_Coils[170]:=FALSE;  //Turbo pump readbacks
mb_Input_Coils[171]:=FALSE;  //Turbo pump readbacks
mb_Input_Coils[172]:=FALSE;  //Turbo pump readbacks
mb_Input_Coils[173]:=FALSE;  //Turbo pump readbacks
mb_Input_Coils[174]:=FALSE;  //Turbo pump readbacks
mb_Input_Coils[175]:=FALSE;  //Turbo pump readbacks
mb_Input_Coils[176]:=FALSE;  //Turbo pump readbacks
mb_Input_Coils[177]:=FALSE;  //Turbo pump readbacks
mb_Input_Coils[178]:=FALSE;  //Turbo pump readbacks
mb_Input_Coils[179]:=FALSE;  //Turbo pump readbacks
mb_Input_Coils[180]:=FALSE;  //Turbo pump readbacks
mb_Input_Coils[181]:=FALSE;  //Turbo pump readbacks
mb_Input_Coils[182]:=FALSE;  //Turbo pump readbacks
mb_Input_Coils[183]:=FALSE;  //Turbo pump readbacks
mb_Input_Coils[184]:=FALSE;  //Turbo pump readbacks
mb_Input_Coils[185]:=FALSE;  //Turbo pump readbacks
mb_Input_Coils[186]:=FALSE;  //Turbo pump readbacks
mb_Input_Coils[187]:=FALSE;  //Turbo pump readbacks
mb_Input_Coils[188]:=FALSE;  //Turbo pump readbacks
mb_Input_Coils[189]:=FALSE;  //Turbo pump readbacks
mb_Input_Coils[190]:=FALSE;  //Turbo pump readbacks
mb_Input_Coils[191]:=FALSE;  //Turbo pump readbacks
mb_Input_Coils[192]:=FALSE;  //Turbo pump readbacks
mb_Input_Coils[193]:=FALSE;  //Turbo pump readbacks
mb_Input_Coils[194]:=FALSE;  //Turbo pump readbacks
mb_Input_Coils[195]:=FALSE;  //Turbo pump readbacks
mb_Input_Coils[196]:=FALSE;  //Turbo pump readbacks
mb_Input_Coils[197]:=FALSE;  //Turbo pump readbacks
mb_Input_Coils[198]:=FALSE;  //Turbo pump readbacks
mb_Input_Coils[199]:=FALSE;  //Turbo pump readbacks
mb_Input_Coils[200]:=FALSE;  //Turbo pump readbacks
mb_Input_Coils[201]:=FALSE;  //Turbo pump readbacks
mb_Input_Coils[202]:=FALSE;  //Turbo pump readbacks
mb_Input_Coils[203]:=FALSE;  //Turbo pump readbacks
mb_Input_Coils[204]:=FALSE;  //Turbo pump readbacks
mb_Input_Coils[205]:=FALSE;  //Turbo pump readbacks
mb_Input_Coils[206]:=FALSE;  //Turbo pump readbacks
mb_Input_Coils[207]:=FALSE;  //Turbo pump readbacks
mb_Input_Coils[208]:=FALSE;  //Turbo pump readbacks
mb_Input_Coils[209]:=FALSE;  //Turbo pump readbacks
mb_Input_Coils[210]:=FALSE;  //Turbo pump readbacks
mb_Input_Coils[211]:=FALSE;  //Turbo pump readbacks
mb_Input_Coils[212]:=FALSE;  //Turbo pump readbacks
mb_Input_Coils[213]:=FALSE;  //Turbo pump readbacks
mb_Input_Coils[214]:=FALSE;  //Turbo pump readbacks
mb_Input_Coils[215]:=FALSE;  //Turbo pump readbacks
mb_Input_Coils[216]:=FALSE;  //Turbo pump readbacks
mb_Input_Coils[217]:=FALSE;  //Turbo pump readbacks
mb_Input_Coils[218]:=FALSE;  //Turbo pump readbacks
mb_Input_Coils[219]:=FALSE;  //Turbo pump readbacks
mb_Input_Coils[220]:=vgPBT_GCC_02.xAT_VAC;  //VG readbacks
mb_Input_Coils[221]:=vgPBT_GCC_02.xHV_DIS;  //VG readbacks
mb_Input_Coils[222]:=vgPBT_GCC_04.xAT_VAC;  //VG readbacks
mb_Input_Coils[223]:=vgPBT_GCC_04.xHV_DIS;  //VG readbacks
mb_Input_Coils[224]:=vgPBT_GCC_06.xAT_VAC;  //VG readbacks
mb_Input_Coils[225]:=vgPBT_GCC_06.xHV_DIS;  //VG readbacks
mb_Input_Coils[226]:=vgPBT_GCC_07.xAT_VAC;  //VG readbacks
mb_Input_Coils[227]:=vgPBT_GCC_07.xHV_DIS;  //VG readbacks
mb_Input_Coils[228]:=vgPBT_GCC_09.xAT_VAC;  //VG readbacks
mb_Input_Coils[229]:=vgPBT_GCC_09.xHV_DIS;  //VG readbacks
mb_Input_Coils[230]:=vgPBT_GCC_02.xPRESS_OK;  //VG readbacks
mb_Input_Coils[231]:=vgPBT_GCC_04.xPRESS_OK;  //VG readbacks
mb_Input_Coils[232]:=vgPBT_GCC_06.xPRESS_OK;  //VG readbacks
mb_Input_Coils[233]:=vgPBT_GCC_07.xPRESS_OK;  //VG readbacks
mb_Input_Coils[234]:=vgPBT_GCC_09.xPRESS_OK;  //VG readbacks
mb_Input_Coils[235]:=FALSE;  //VG readbacks
mb_Input_Coils[236]:=FALSE;  //VG readbacks
mb_Input_Coils[237]:=FALSE;  //VG readbacks
mb_Input_Coils[238]:=FALSE;  //VG readbacks
mb_Input_Coils[239]:=FALSE;  //VG readbacks
mb_Input_Coils[240]:=FALSE;  //VG readbacks
mb_Input_Coils[241]:=FALSE;  //VG readbacks
mb_Input_Coils[242]:=FALSE;  //VG readbacks
mb_Input_Coils[243]:=FALSE;  //VG readbacks
mb_Input_Coils[244]:=FALSE;  //VG readbacks
mb_Input_Coils[245]:=FALSE;  //VG readbacks
mb_Input_Coils[246]:=FALSE;  //VG readbacks
mb_Input_Coils[247]:=FALSE;  //VG readbacks
mb_Input_Coils[248]:=FALSE;  //VG readbacks
mb_Input_Coils[249]:=FALSE;  //VG readbacks
mb_Input_Coils[250]:=FALSE;  //VG readbacks
mb_Input_Coils[251]:=FALSE;  //VG readbacks
mb_Input_Coils[252]:=FALSE;  //VG readbacks
mb_Input_Coils[253]:=FALSE;  //VG readbacks
mb_Input_Coils[254]:=FALSE;  //VG readbacks
mb_Input_Coils[255]:=FALSE;  //VG readbacks

END_PROGRAM

// ---- POUs/Modbus/p_ModbusTx_InputReg.TcPOU
PROGRAM p_ModbusTx_InputReg
VAR
END_VAR

mb_Input_Registers[0]:=0;  //System info
mb_Input_Registers[1]:=0;  //System info
mb_Input_Registers[2]:=0;  //System info
mb_Input_Registers[3]:=0;  //System info
mb_Input_Registers[4]:=0;  //System info
mb_Input_Registers[5]:=0;  //System info
mb_Input_Registers[6]:=0;  //System info
mb_Input_Registers[7]:=0;  //System info
mb_Input_Registers[8]:=0;  //System info
mb_Input_Registers[9]:=0;  //System info
mb_Input_Registers[10]:=0;  //VG pressure readbacks
mb_Input_Registers[11]:=0;  //VG pressure readbacks
mb_Input_Registers[12]:=0;  //VG pressure readbacks
mb_Input_Registers[13]:=0;  //VG pressure readbacks
mb_Input_Registers[14]:=0;  //VG pressure readbacks
mb_Input_Registers[15]:=0;  //VG pressure readbacks
mb_Input_Registers[16]:=0;  //VG pressure readbacks
mb_Input_Registers[17]:=0;  //VG pressure readbacks
mb_Input_Registers[18]:=0;  //VG pressure readbacks
mb_Input_Registers[19]:=0;  //VG pressure readbacks
mb_Input_Registers[20]:=0;  //VG pressure readbacks
mb_Input_Registers[21]:=0;  //VG pressure readbacks
mb_Input_Registers[22]:=0;  //VG pressure readbacks
mb_Input_Registers[23]:=0;  //VG pressure readbacks
mb_Input_Registers[24]:=0;  //VG pressure readbacks
mb_Input_Registers[25]:=0;  //VG pressure readbacks
mb_Input_Registers[26]:=0;  //VG pressure readbacks
mb_Input_Registers[27]:=0;  //VG pressure readbacks
mb_Input_Registers[28]:=0;  //VG pressure readbacks
mb_Input_Registers[29]:=0;  //VG pressure readbacks
mb_Input_Registers[30]:=0;  //VG pressure readbacks
mb_Input_Registers[31]:=0;  //VG pressure readbacks
mb_Input_Registers[32]:=0;  //VG pressure readbacks
mb_Input_Registers[33]:=0;  //VG pressure readbacks
mb_Input_Registers[34]:=0;  //VG pressure readbacks
mb_Input_Registers[35]:=0;  //VG pressure readbacks
mb_Input_Registers[36]:=0;  //VG pressure readbacks
mb_Input_Registers[37]:=0;  //VG pressure readbacks
mb_Input_Registers[38]:=0;  //VG pressure readbacks
mb_Input_Registers[39]:=0;  //VG pressure readbacks
mb_Input_Registers[40]:=0;  //VG pressure readbacks
mb_Input_Registers[41]:=0;  //VG pressure readbacks
mb_Input_Registers[42]:=0;  //VG pressure readbacks
mb_Input_Registers[43]:=0;  //VG pressure readbacks
mb_Input_Registers[44]:=0;  //VG pressure readbacks
mb_Input_Registers[45]:=0;  //VG pressure readbacks
mb_Input_Registers[46]:=0;  //VG pressure readbacks
mb_Input_Registers[47]:=0;  //VG pressure readbacks
mb_Input_Registers[48]:=0;  //VG pressure readbacks
mb_Input_Registers[49]:=0;  //VG pressure readbacks
mb_Input_Registers[50]:=0;  //VG pressure readbacks
mb_Input_Registers[51]:=0;  //VG pressure readbacks
mb_Input_Registers[52]:=0;  //VG pressure readbacks
mb_Input_Registers[53]:=0;  //VG pressure readbacks
mb_Input_Registers[54]:=0;  //VG pressure readbacks
mb_Input_Registers[55]:=0;  //VG pressure readbacks
mb_Input_Registers[56]:=0;  //VG pressure readbacks
mb_Input_Registers[57]:=0;  //VG pressure readbacks
mb_Input_Registers[58]:=0;  //VG pressure readbacks
mb_Input_Registers[59]:=0;  //VG pressure readbacks
mb_Input_Registers[60]:=0;  //VG pressure readbacks
mb_Input_Registers[61]:=0;  //VG pressure readbacks
mb_Input_Registers[62]:=0;  //VG pressure readbacks
mb_Input_Registers[63]:=0;  //VG pressure readbacks
mb_Input_Registers[64]:=0;  //VG pressure readbacks
mb_Input_Registers[65]:=0;  //VG pressure readbacks
mb_Input_Registers[66]:=0;  //VG pressure readbacks
mb_Input_Registers[67]:=0;  //VG pressure readbacks
mb_Input_Registers[68]:=0;  //VG pressure readbacks
mb_Input_Registers[69]:=0;  //VG pressure readbacks
mb_Input_Registers[70]:=TO_WORD(vgPBT_GPI_02.eState);  //VG state readbacks
mb_Input_Registers[71]:=TO_WORD(vgPBT_GPI_04.eState);  //VG state readbacks
mb_Input_Registers[72]:=TO_WORD(vgPBT_GPI_06.eState);  //VG state readbacks
mb_Input_Registers[73]:=TO_WORD(vgPBT_GPI_07.eState);  //VG state readbacks
mb_Input_Registers[74]:=TO_WORD(vgPBT_GPI_09.eState);  //VG state readbacks
mb_Input_Registers[75]:=TO_WORD(vgPBT_GCC_02.eState);  //VG state readbacks
mb_Input_Registers[76]:=TO_WORD(vgPBT_GCC_04.eState);  //VG state readbacks
mb_Input_Registers[77]:=TO_WORD(vgPBT_GCC_06.eState);  //VG state readbacks
mb_Input_Registers[78]:=TO_WORD(vgPBT_GCC_07.eState);  //VG state readbacks
mb_Input_Registers[79]:=TO_WORD(vgPBT_GCC_09.eState);  //VG state readbacks
mb_Input_Registers[80]:=0;  //VG state readbacks
mb_Input_Registers[81]:=0;  //VG state readbacks
mb_Input_Registers[82]:=0;  //VG state readbacks
mb_Input_Registers[83]:=0;  //VG state readbacks
mb_Input_Registers[84]:=0;  //VG state readbacks
mb_Input_Registers[85]:=0;  //VG state readbacks
mb_Input_Registers[86]:=0;  //VG state readbacks
mb_Input_Registers[87]:=0;  //VG state readbacks
mb_Input_Registers[88]:=0;  //VG state readbacks
mb_Input_Registers[89]:=0;  //VG state readbacks
mb_Input_Registers[90]:=0;  //VG state readbacks
mb_Input_Registers[91]:=0;  //VG state readbacks
mb_Input_Registers[92]:=0;  //VG state readbacks
mb_Input_Registers[93]:=0;  //VG state readbacks
mb_Input_Registers[94]:=0;  //VG state readbacks
mb_Input_Registers[95]:=0;  //VG state readbacks
mb_Input_Registers[96]:=0;  //VG state readbacks
mb_Input_Registers[97]:=0;  //VG state readbacks
mb_Input_Registers[98]:=0;  //VG state readbacks
mb_Input_Registers[99]:=0;  //VG state readbacks
mb_Input_Registers[100]:=0;  //VG state readbacks
mb_Input_Registers[101]:=0;  //VG state readbacks
mb_Input_Registers[102]:=0;  //VG state readbacks
mb_Input_Registers[103]:=0;  //VG state readbacks
mb_Input_Registers[104]:=0;  //VG state readbacks
mb_Input_Registers[105]:=0;  //VG state readbacks
mb_Input_Registers[106]:=0;  //VG state readbacks
mb_Input_Registers[107]:=0;  //VG state readbacks
mb_Input_Registers[108]:=0;  //VG state readbacks
mb_Input_Registers[109]:=0;  //VG state readbacks
mb_Input_Registers[110]:=0;  //VG state readbacks
mb_Input_Registers[111]:=0;  //VG state readbacks
mb_Input_Registers[112]:=0;  //VG state readbacks
mb_Input_Registers[113]:=0;  //VG state readbacks
mb_Input_Registers[114]:=0;  //VG state readbacks
mb_Input_Registers[115]:=0;  //VG state readbacks
mb_Input_Registers[116]:=0;  //VG state readbacks
mb_Input_Registers[117]:=0;  //VG state readbacks
mb_Input_Registers[118]:=0;  //VG state readbacks
mb_Input_Registers[119]:=0;  //VG state readbacks
mb_Input_Registers[120]:=0;  //default
mb_Input_Registers[121]:=0;  //default
mb_Input_Registers[122]:=0;  //default
mb_Input_Registers[123]:=0;  //default
mb_Input_Registers[124]:=0;  //default
mb_Input_Registers[125]:=0;  //default
mb_Input_Registers[126]:=0;  //default
mb_Input_Registers[127]:=0;  //default
mb_Input_Registers[128]:=0;  //default
mb_Input_Registers[129]:=0;  //default
mb_Input_Registers[130]:=0;  //default
mb_Input_Registers[131]:=0;  //default
mb_Input_Registers[132]:=0;  //default
mb_Input_Registers[133]:=0;  //default
mb_Input_Registers[134]:=0;  //default
mb_Input_Registers[135]:=0;  //default
mb_Input_Registers[136]:=0;  //default
mb_Input_Registers[137]:=0;  //default
mb_Input_Registers[138]:=0;  //default
mb_Input_Registers[139]:=0;  //default
mb_Input_Registers[140]:=0;  //default
mb_Input_Registers[141]:=0;  //default
mb_Input_Registers[142]:=0;  //default
mb_Input_Registers[143]:=0;  //default
mb_Input_Registers[144]:=0;  //default
mb_Input_Registers[145]:=0;  //default
mb_Input_Registers[146]:=0;  //default
mb_Input_Registers[147]:=0;  //default
mb_Input_Registers[148]:=0;  //default
mb_Input_Registers[149]:=0;  //default
mb_Input_Registers[150]:=0;  //default
mb_Input_Registers[151]:=0;  //default
mb_Input_Registers[152]:=0;  //default
mb_Input_Registers[153]:=0;  //default
mb_Input_Registers[154]:=0;  //default
mb_Input_Registers[155]:=0;  //default
mb_Input_Registers[156]:=0;  //default
mb_Input_Registers[157]:=0;  //default
mb_Input_Registers[158]:=0;  //default
mb_Input_Registers[159]:=0;  //default
mb_Input_Registers[160]:=0;  //default
mb_Input_Registers[161]:=0;  //default
mb_Input_Registers[162]:=0;  //default
mb_Input_Registers[163]:=0;  //default
mb_Input_Registers[164]:=0;  //default
mb_Input_Registers[165]:=0;  //default
mb_Input_Registers[166]:=0;  //default
mb_Input_Registers[167]:=0;  //default
mb_Input_Registers[168]:=0;  //default
mb_Input_Registers[169]:=0;  //default
mb_Input_Registers[170]:=0;  //default
mb_Input_Registers[171]:=0;  //default
mb_Input_Registers[172]:=0;  //default
mb_Input_Registers[173]:=0;  //default
mb_Input_Registers[174]:=0;  //default
mb_Input_Registers[175]:=0;  //default
mb_Input_Registers[176]:=0;  //default
mb_Input_Registers[177]:=0;  //default
mb_Input_Registers[178]:=0;  //default
mb_Input_Registers[179]:=0;  //default
mb_Input_Registers[180]:=0;  //default
mb_Input_Registers[181]:=0;  //default
mb_Input_Registers[182]:=0;  //default
mb_Input_Registers[183]:=0;  //default
mb_Input_Registers[184]:=0;  //default
mb_Input_Registers[185]:=0;  //default
mb_Input_Registers[186]:=0;  //default
mb_Input_Registers[187]:=0;  //default
mb_Input_Registers[188]:=0;  //default
mb_Input_Registers[189]:=0;  //default
mb_Input_Registers[190]:=0;  //default
mb_Input_Registers[191]:=0;  //default
mb_Input_Registers[192]:=0;  //default
mb_Input_Registers[193]:=0;  //default
mb_Input_Registers[194]:=0;  //default
mb_Input_Registers[195]:=0;  //default
mb_Input_Registers[196]:=0;  //default
mb_Input_Registers[197]:=0;  //default
mb_Input_Registers[198]:=0;  //default
mb_Input_Registers[199]:=0;  //default
mb_Input_Registers[200]:=0;  //default
mb_Input_Registers[201]:=0;  //default
mb_Input_Registers[202]:=0;  //default
mb_Input_Registers[203]:=0;  //default
mb_Input_Registers[204]:=0;  //default
mb_Input_Registers[205]:=0;  //default
mb_Input_Registers[206]:=0;  //default
mb_Input_Registers[207]:=0;  //default
mb_Input_Registers[208]:=0;  //default
mb_Input_Registers[209]:=0;  //default
mb_Input_Registers[210]:=0;  //default
mb_Input_Registers[211]:=0;  //default
mb_Input_Registers[212]:=0;  //default
mb_Input_Registers[213]:=0;  //default
mb_Input_Registers[214]:=0;  //default
mb_Input_Registers[215]:=0;  //default
mb_Input_Registers[216]:=0;  //default
mb_Input_Registers[217]:=0;  //default
mb_Input_Registers[218]:=0;  //default
mb_Input_Registers[219]:=0;  //default
mb_Input_Registers[220]:=0;  //default
mb_Input_Registers[221]:=0;  //default
mb_Input_Registers[222]:=0;  //default
mb_Input_Registers[223]:=0;  //default
mb_Input_Registers[224]:=0;  //default
mb_Input_Registers[225]:=0;  //default
mb_Input_Registers[226]:=0;  //default
mb_Input_Registers[227]:=0;  //default
mb_Input_Registers[228]:=0;  //default
mb_Input_Registers[229]:=0;  //default
mb_Input_Registers[230]:=0;  //default
mb_Input_Registers[231]:=0;  //default
mb_Input_Registers[232]:=0;  //default
mb_Input_Registers[233]:=0;  //default
mb_Input_Registers[234]:=0;  //default
mb_Input_Registers[235]:=0;  //default
mb_Input_Registers[236]:=0;  //default
mb_Input_Registers[237]:=0;  //default
mb_Input_Registers[238]:=0;  //default
mb_Input_Registers[239]:=0;  //default
mb_Input_Registers[240]:=0;  //default
mb_Input_Registers[241]:=0;  //default
mb_Input_Registers[242]:=0;  //default
mb_Input_Registers[243]:=0;  //default
mb_Input_Registers[244]:=0;  //default
mb_Input_Registers[245]:=0;  //default
mb_Input_Registers[246]:=0;  //default
mb_Input_Registers[247]:=0;  //default
mb_Input_Registers[248]:=0;  //default
mb_Input_Registers[249]:=0;  //default
mb_Input_Registers[250]:=0;  //default
mb_Input_Registers[251]:=0;  //default
mb_Input_Registers[252]:=0;  //default
mb_Input_Registers[253]:=0;  //default
mb_Input_Registers[254]:=0;  //default
mb_Input_Registers[255]:=0;  //default

END_PROGRAM

// ---- POUs/Modbus/p_ModbusTx_OutputCoils.TcPOU
PROGRAM p_ModbusTx_OutputCoils
VAR
END_VAR

mb_Output_Coils[0]:=FALSE;  //System Controls
mb_Output_Coils[1]:=g_stSystem.xOverrideMode;  //System Controls
mb_Output_Coils[2]:=FALSE;  //System Controls
mb_Output_Coils[3] :=q_xXCS_VGC_OK;  //System Controls
mb_Output_Coils[4] :=FALSE;  //System Controls
mb_Output_Coils[5] :=q_xXCS_MPSOK;  //System Controlsmb_Output_Coils[2]:=FALSE;  //System Controls
mb_Output_Coils[6]:=FALSE;  //System Controls
mb_Output_Coils[7]:=FALSE;  //System Controls
mb_Output_Coils[8]:=FALSE;  //System Controls
mb_Output_Coils[9]:=FALSE;  //System Controls
mb_Output_Coils[10]:=vgcPBT_VGC_01.xOPN_SW;  //Valve switch controls
mb_Output_Coils[11]:=vgcPBT_VGC_02.xOPN_SW;  //Valve switch controls
mb_Output_Coils[12]:=vgcPBT_VGC_03.xOPN_SW;  //Valve switch controls
mb_Output_Coils[13]:=vgcPBT_VGC_04.xOPN_SW;  //Valve switch controls
mb_Output_Coils[14]:=FALSE;  //Valve switch controls
mb_Output_Coils[15]:=FALSE;  //Valve switch controls
mb_Output_Coils[16]:=FALSE;  //Valve switch controls
mb_Output_Coils[17]:=FALSE;  //Valve switch controls
mb_Output_Coils[18]:=FALSE;  //Valve switch controls
mb_Output_Coils[19]:=FALSE;  //Valve switch controls
mb_Output_Coils[20]:=FALSE;  //Valve switch controls
mb_Output_Coils[21]:=FALSE;  //Valve switch controls
mb_Output_Coils[22]:=FALSE;  //Valve switch controls
mb_Output_Coils[23]:=FALSE;  //Valve switch controls
mb_Output_Coils[24]:=FALSE;  //Valve switch controls
mb_Output_Coils[25]:=FALSE;  //Valve switch controls
mb_Output_Coils[26]:=FALSE;  //Valve switch controls
mb_Output_Coils[27]:=FALSE;  //Valve switch controls
mb_Output_Coils[28]:=FALSE;  //Valve switch controls
mb_Output_Coils[29]:=FALSE;  //Valve switch controls
mb_Output_Coils[30]:=FALSE;  //Valve switch controls
mb_Output_Coils[31]:=FALSE;  //Valve switch controls
mb_Output_Coils[32]:=FALSE;  //Valve switch controls
mb_Output_Coils[33]:=FALSE;  //Valve switch controls
mb_Output_Coils[34]:=FALSE;  //Valve switch controls
mb_Output_Coils[35]:=FALSE;  //Valve switch controls
mb_Output_Coils[36]:=FALSE;  //Valve switch controls
mb_Output_Coils[37]:=FALSE;  //Valve switch controls
mb_Output_Coils[38]:=FALSE;  //Valve switch controls
mb_Output_Coils[39]:=FALSE;  //Valve switch controls
mb_Output_Coils[40]:=FALSE;  //Valve switch controls
mb_Output_Coils[41]:=FALSE;  //Valve switch controls
mb_Output_Coils[42]:=FALSE;  //Valve switch controls
mb_Output_Coils[43]:=FALSE;  //Valve switch controls
mb_Output_Coils[44]:=FALSE;  //Valve switch controls
mb_Output_Coils[45]:=FALSE;  //Valve switch controls
mb_Output_Coils[46]:=FALSE;  //Valve switch controls
mb_Output_Coils[47]:=FALSE;  //Valve switch controls
mb_Output_Coils[48]:=FALSE;  //Valve switch controls
mb_Output_Coils[49]:=FALSE;  //Valve switch controls
mb_Output_Coils[50]:=FALSE;  //Valve switch controls
mb_Output_Coils[51]:=FALSE;  //Valve switch controls
mb_Output_Coils[52]:=FALSE;  //Valve switch controls
mb_Output_Coils[53]:=FALSE;  //Valve switch controls
mb_Output_Coils[54]:=FALSE;  //Valve switch controls
mb_Output_Coils[55]:=FALSE;  //Valve switch controls
mb_Output_Coils[56]:=FALSE;  //Valve switch controls
mb_Output_Coils[57]:=FALSE;  //Valve switch controls
mb_Output_Coils[58]:=FALSE;  //Valve switch controls
mb_Output_Coils[59]:=FALSE;  //Valve switch controls
mb_Output_Coils[60]:=FALSE;  //Valve switch controls
mb_Output_Coils[61]:=FALSE;  //Valve switch controls
mb_Output_Coils[62]:=FALSE;  //Valve switch controls
mb_Output_Coils[63]:=FALSE;  //Valve switch controls
mb_Output_Coils[64]:=FALSE;  //Valve switch controls
mb_Output_Coils[65]:=FALSE;  //Valve switch controls
mb_Output_Coils[66]:=FALSE;  //Valve switch controls
mb_Output_Coils[67]:=FALSE;  //Valve switch controls
mb_Output_Coils[68]:=FALSE;  //Valve switch controls
mb_Output_Coils[69]:=FALSE;  //Valve switch controls
mb_Output_Coils[70]:=FALSE;  //Turbo Controls
mb_Output_Coils[71]:=FALSE;  //Turbo Controls
mb_Output_Coils[72]:=FALSE;  //Turbo Controls
mb_Output_Coils[74]:=FALSE;  //Turbo Controls
mb_Output_Coils[75]:=FALSE;  //Turbo Controls
mb_Output_Coils[76]:=FALSE;  //Turbo Controls
mb_Output_Coils[77]:=FALSE;  //Turbo Controls
mb_Output_Coils[78]:=FALSE;  //Turbo Controls
mb_Output_Coils[79]:=FALSE;  //Turbo Controls
mb_Output_Coils[80]:=FALSE;  //Turbo Controls
mb_Output_Coils[81]:=FALSE;  //Turbo Controls
mb_Output_Coils[82]:=FALSE;  //Turbo Controls
mb_Output_Coils[83]:=FALSE;  //Turbo Controls
mb_Output_Coils[84]:=FALSE;  //Turbo Controls
mb_Output_Coils[85]:=FALSE;  //Turbo Controls
mb_Output_Coils[86]:=FALSE;  //Turbo Controls
mb_Output_Coils[87]:=FALSE;  //Turbo Controls
mb_Output_Coils[88]:=FALSE;  //Turbo Controls
mb_Output_Coils[89]:=FALSE;  //Turbo Controls
mb_Output_Coils[90]:=FALSE;  //Turbo Controls
mb_Output_Coils[91]:=FALSE;  //Turbo Controls
mb_Output_Coils[92]:=FALSE;  //Turbo Controls
mb_Output_Coils[93]:=FALSE;  //Turbo Controls
mb_Output_Coils[94]:=FALSE;  //Turbo Controls
mb_Output_Coils[95]:=FALSE;  //Turbo Controls
mb_Output_Coils[96]:=FALSE;  //Turbo Controls
mb_Output_Coils[97]:=FALSE;  //Turbo Controls
mb_Output_Coils[98]:=FALSE;  //Turbo Controls
mb_Output_Coils[99]:=FALSE;  //Turbo Controls
mb_Output_Coils[100]:=FALSE;  //Turbo Controls
mb_Output_Coils[101]:=FALSE;  //Turbo Controls
mb_Output_Coils[102]:=FALSE;  //Turbo Controls
mb_Output_Coils[103]:=FALSE;  //Turbo Controls
mb_Output_Coils[104]:=FALSE;  //Turbo Controls
mb_Output_Coils[105]:=FALSE;  //Turbo Controls
mb_Output_Coils[106]:=FALSE;  //Turbo Controls
mb_Output_Coils[107]:=FALSE;  //Turbo Controls
mb_Output_Coils[108]:=FALSE;  //Turbo Controls
mb_Output_Coils[109]:=FALSE;  //Turbo Controls
mb_Output_Coils[110]:=FALSE;  //Turbo Controls
mb_Output_Coils[111]:=FALSE;  //Turbo Controls
mb_Output_Coils[112]:=FALSE;  //Turbo Controls
mb_Output_Coils[113]:=FALSE;  //Turbo Controls
mb_Output_Coils[114]:=FALSE;  //Turbo Controls
mb_Output_Coils[115]:=FALSE;  //Turbo Controls
mb_Output_Coils[116]:=FALSE;  //Turbo Controls
mb_Output_Coils[117]:=FALSE;  //Turbo Controls
mb_Output_Coils[118]:=FALSE;  //Turbo Controls
mb_Output_Coils[119]:=FALSE;  //Turbo Controls
mb_Output_Coils[120]:=vgPBT_GCC_02.xHV_SW;  //CC HV Enable
mb_Output_Coils[121]:=vgPBT_GCC_04.xHV_SW;  //CC HV Enable
mb_Output_Coils[122]:=vgPBT_GCC_06.xHV_SW;  //CC HV Enable
mb_Output_Coils[123]:=vgPBT_GCC_07.xHV_SW;  //CC HV Enable
mb_Output_Coils[124]:=vgPBT_GCC_09.xHV_SW;  //CC HV Enable
mb_Output_Coils[125]:=FALSE;  //CC HV Enable
mb_Output_Coils[126]:=FALSE;  //CC HV Enable
mb_Output_Coils[127]:=FALSE;  //CC HV Enable
mb_Output_Coils[128]:=FALSE;  //CC HV Enable
mb_Output_Coils[129]:=FALSE;  //CC HV Enable
mb_Output_Coils[130]:=FALSE;  //CC HV Enable
mb_Output_Coils[131]:=FALSE;  //CC HV Enable
mb_Output_Coils[132]:=FALSE;  //CC HV Enable
mb_Output_Coils[133]:=FALSE;  //CC HV Enable
mb_Output_Coils[134]:=FALSE;  //CC HV Enable
mb_Output_Coils[135]:=FALSE;  //CC HV Enable
mb_Output_Coils[136]:=FALSE;  //CC HV Enable
mb_Output_Coils[137]:=FALSE;  //CC HV Enable
mb_Output_Coils[138]:=FALSE;  //CC HV Enable
mb_Output_Coils[139]:=FALSE;  //CC HV Enable
mb_Output_Coils[140]:=FALSE;  //CC HV Enable
mb_Output_Coils[141]:=FALSE;  //CC HV Enable
mb_Output_Coils[142]:=FALSE;  //CC HV Enable
mb_Output_Coils[143]:=FALSE;  //CC HV Enable
mb_Output_Coils[144]:=FALSE;  //CC HV Enable
mb_Output_Coils[145]:=FALSE;  //CC HV Enable
mb_Output_Coils[146]:=FALSE;  //CC HV Enable
mb_Output_Coils[147]:=FALSE;  //CC HV Enable
mb_Output_Coils[148]:=FALSE;  //CC HV Enable
mb_Output_Coils[149]:=FALSE;  //CC HV Enable
mb_Output_Coils[150]:=FALSE;  //CC HV Enable
mb_Output_Coils[151]:=FALSE;  //CC HV Enable
mb_Output_Coils[152]:=FALSE;  //CC HV Enable
mb_Output_Coils[153]:=FALSE;  //CC HV Enable
mb_Output_Coils[154]:=FALSE;  //CC HV Enable
mb_Output_Coils[155]:=FALSE;  //CC HV Enable
mb_Output_Coils[156]:=FALSE;  //CC HV Enable
mb_Output_Coils[157]:=FALSE;  //CC HV Enable
mb_Output_Coils[158]:=FALSE;  //CC HV Enable
mb_Output_Coils[159]:=FALSE;  //CC HV Enable
mb_Output_Coils[160]:=FALSE;  //
mb_Output_Coils[161]:=FALSE;  //
mb_Output_Coils[162]:=FALSE;  //
mb_Output_Coils[163]:=FALSE;  //
mb_Output_Coils[164]:=FALSE;  //
mb_Output_Coils[165]:=FALSE;  //
mb_Output_Coils[166]:=FALSE;  //
mb_Output_Coils[167]:=FALSE;  //
mb_Output_Coils[168]:=FALSE;  //
mb_Output_Coils[169]:=FALSE;  //
mb_Output_Coils[170]:=FALSE;  //
mb_Output_Coils[171]:=FALSE;  //
mb_Output_Coils[172]:=FALSE;  //
mb_Output_Coils[173]:=FALSE;  //
mb_Output_Coils[174]:=FALSE;  //
mb_Output_Coils[175]:=FALSE;  //
mb_Output_Coils[176]:=FALSE;  //
mb_Output_Coils[177]:=FALSE;  //
mb_Output_Coils[178]:=FALSE;  //
mb_Output_Coils[179]:=FALSE;  //
mb_Output_Coils[180]:=FALSE;  //
mb_Output_Coils[181]:=FALSE;  //
mb_Output_Coils[182]:=FALSE;  //
mb_Output_Coils[183]:=FALSE;  //
mb_Output_Coils[184]:=FALSE;  //
mb_Output_Coils[185]:=FALSE;  //
mb_Output_Coils[186]:=FALSE;  //
mb_Output_Coils[187]:=FALSE;  //
mb_Output_Coils[188]:=FALSE;  //
mb_Output_Coils[189]:=FALSE;  //
mb_Output_Coils[190]:=FALSE;  //
mb_Output_Coils[191]:=FALSE;  //
mb_Output_Coils[192]:=FALSE;  //
mb_Output_Coils[193]:=FALSE;  //
mb_Output_Coils[194]:=FALSE;  //
mb_Output_Coils[195]:=FALSE;  //
mb_Output_Coils[196]:=FALSE;  //
mb_Output_Coils[197]:=FALSE;  //
mb_Output_Coils[198]:=FALSE;  //
mb_Output_Coils[199]:=FALSE;  //
mb_Output_Coils[200]:=vgcPBT_VGC_01.xOvrdOpn;  //Valve overrides
mb_Output_Coils[201]:=vgcPBT_VGC_02.xOvrdOpn;  //Valve overrides
mb_Output_Coils[202]:=vgcPBT_VGC_03.xOvrdOpn;  //Valve overrides
mb_Output_Coils[203]:=vgcPBT_VGC_04.xOvrdOpn;  //Valve overrides
mb_Output_Coils[204]:=FALSE;  //
mb_Output_Coils[205]:=FALSE;  //
mb_Output_Coils[206]:=FALSE;  //
mb_Output_Coils[207]:=FALSE;  //
mb_Output_Coils[208]:=FALSE;  //
mb_Output_Coils[209]:=FALSE;  //
mb_Output_Coils[210]:=FALSE;  //
mb_Output_Coils[211]:=FALSE;  //
mb_Output_Coils[212]:=FALSE;  //
mb_Output_Coils[213]:=FALSE;  //
mb_Output_Coils[214]:=FALSE;  //
mb_Output_Coils[215]:=FALSE;  //
mb_Output_Coils[216]:=FALSE;  //
mb_Output_Coils[217]:=FALSE;  //
mb_Output_Coils[218]:=FALSE;  //
mb_Output_Coils[219]:=FALSE;  //
mb_Output_Coils[220]:=FALSE;  //
mb_Output_Coils[221]:=FALSE;  //
mb_Output_Coils[222]:=FALSE;  //
mb_Output_Coils[223]:=FALSE;  //
mb_Output_Coils[224]:=FALSE;  //
mb_Output_Coils[225]:=FALSE;  //
mb_Output_Coils[226]:=FALSE;  //
mb_Output_Coils[227]:=FALSE;  //
mb_Output_Coils[228]:=FALSE;  //
mb_Output_Coils[229]:=FALSE;  //
mb_Output_Coils[230]:=FALSE;  //
mb_Output_Coils[231]:=FALSE;  //
mb_Output_Coils[232]:=FALSE;  //
mb_Output_Coils[233]:=FALSE;  //
mb_Output_Coils[234]:=FALSE;  //
mb_Output_Coils[235]:=FALSE;  //
mb_Output_Coils[236]:=FALSE;  //
mb_Output_Coils[237]:=FALSE;  //
mb_Output_Coils[238]:=FALSE;  //
mb_Output_Coils[239]:=FALSE;  //
mb_Output_Coils[240]:=FALSE;  //
mb_Output_Coils[241]:=FALSE;  //
mb_Output_Coils[242]:=FALSE;  //
mb_Output_Coils[243]:=FALSE;  //
mb_Output_Coils[244]:=FALSE;  //
mb_Output_Coils[245]:=FALSE;  //
mb_Output_Coils[246]:=FALSE;  //
mb_Output_Coils[247]:=FALSE;  //
mb_Output_Coils[248]:=FALSE;  //
mb_Output_Coils[249]:=FALSE;  //
mb_Output_Coils[250]:=FALSE;  //
mb_Output_Coils[251]:=FALSE;  //
mb_Output_Coils[252]:=FALSE;  //
mb_Output_Coils[253]:=FALSE;  //
mb_Output_Coils[254]:=FALSE;  //
mb_Output_Coils[255]:=FALSE;  //

END_PROGRAM

// ---- POUs/Modbus/p_ModbusTx_OutputReg.TcPOU
PROGRAM p_ModbusTx_OutputReg
VAR
END_VAR

mb_Output_Registers[0]:=0;  //System parameters
mb_Output_Registers[1]:=0;  //System parameters
mb_Output_Registers[2]:=0;  //System parameters
mb_Output_Registers[3]:=0;  //System parameters
mb_Output_Registers[4]:=0;  //System parameters
mb_Output_Registers[5]:=0;  //System parameters
mb_Output_Registers[6]:=0;  //System parameters
mb_Output_Registers[7]:=0;  //System parameters
mb_Output_Registers[8]:=0;  //System parameters
mb_Output_Registers[9]:=0;  //System parameters
(*mb_Output_Registers[10]:=vgPBT_GCC_02.iVacSp;  //VG setpoint
mb_Output_Registers[11]:=vgPBT_GPI_02.iVacSp;  //VG setpoint
mb_Output_Registers[12]:=vgPBT_GCC_04.iVacSp;  //VG setpoint
mb_Output_Registers[13]:=vgPBT_GPI_04.iVacSp;  //VG setpoint
mb_Output_Registers[14]:=vgPBT_GCC_06.iVacSp;  //VG setpoint
mb_Output_Registers[15]:=vgPBT_GPI_06.iVacSp;  //VG setpoint
mb_Output_Registers[16]:=vgPBT_GCC_07.iVacSp;  //VG setpoint
mb_Output_Registers[17]:=vgPBT_GPI_07.iVacSp;  //VG setpoint
mb_Output_Registers[18]:=vgPBT_GCC_09.iVacSp;  //VG setpoint
mb_Output_Registers[19]:=vgPBT_GPI_09.iVacSp;  //VG setpoint*)
mb_Output_Registers[20]:=0;  //VG setpoint
mb_Output_Registers[21]:=0;  //VG setpoint
mb_Output_Registers[22]:=0;  //VG setpoint
mb_Output_Registers[23]:=0;  //VG setpoint
mb_Output_Registers[24]:=0;  //VG setpoint
mb_Output_Registers[25]:=0;  //VG setpoint
mb_Output_Registers[26]:=0;  //VG setpoint
mb_Output_Registers[27]:=0;  //VG setpoint
mb_Output_Registers[28]:=0;  //VG setpoint
mb_Output_Registers[29]:=0;  //VG setpoint
mb_Output_Registers[30]:=0;  //VG setpoint
mb_Output_Registers[31]:=0;  //VG setpoint
mb_Output_Registers[32]:=0;  //VG setpoint
mb_Output_Registers[33]:=0;  //VG setpoint
mb_Output_Registers[34]:=0;  //VG setpoint
mb_Output_Registers[35]:=0;  //VG setpoint
mb_Output_Registers[36]:=0;  //VG setpoint
mb_Output_Registers[37]:=0;  //VG setpoint
mb_Output_Registers[38]:=0;  //VG setpoint
mb_Output_Registers[39]:=0;  //VG setpoint
mb_Output_Registers[40]:=0;  //VG setpoint
mb_Output_Registers[41]:=0;  //VG setpoint
mb_Output_Registers[42]:=0;  //VG setpoint
mb_Output_Registers[43]:=0;  //VG setpoint
mb_Output_Registers[44]:=0;  //VG setpoint
mb_Output_Registers[45]:=0;  //VG setpoint
mb_Output_Registers[46]:=0;  //VG setpoint
mb_Output_Registers[47]:=0;  //VG setpoint
mb_Output_Registers[48]:=0;  //VG setpoint
mb_Output_Registers[49]:=0;  //VG setpoint
mb_Output_Registers[50]:=0;  //VG setpoint
mb_Output_Registers[51]:=0;  //VG setpoint
mb_Output_Registers[52]:=0;  //VG setpoint
mb_Output_Registers[53]:=0;  //VG setpoint
mb_Output_Registers[54]:=0;  //VG setpoint
mb_Output_Registers[55]:=0;  //VG setpoint
mb_Output_Registers[56]:=0;  //VG setpoint
mb_Output_Registers[57]:=0;  //VG setpoint
mb_Output_Registers[58]:=0;  //VG setpoint
mb_Output_Registers[59]:=0;  //VG setpoint
mb_Output_Registers[60]:=0;  //default
mb_Output_Registers[61]:=0;  //default
mb_Output_Registers[62]:=0;  //default
mb_Output_Registers[63]:=0;  //default
mb_Output_Registers[64]:=0;  //default
mb_Output_Registers[65]:=0;  //default
mb_Output_Registers[66]:=0;  //default
mb_Output_Registers[67]:=0;  //default
mb_Output_Registers[68]:=0;  //default
mb_Output_Registers[69]:=0;  //default
mb_Output_Registers[70]:=0;  //default
mb_Output_Registers[71]:=0;  //default
mb_Output_Registers[72]:=0;  //default
mb_Output_Registers[73]:=0;  //default
mb_Output_Registers[74]:=0;  //default
mb_Output_Registers[75]:=0;  //default
mb_Output_Registers[76]:=0;  //default
mb_Output_Registers[77]:=0;  //default
mb_Output_Registers[78]:=0;  //default
mb_Output_Registers[79]:=0;  //default
mb_Output_Registers[80]:=0;  //default
mb_Output_Registers[81]:=0;  //default
mb_Output_Registers[82]:=0;  //default
mb_Output_Registers[83]:=0;  //default
mb_Output_Registers[84]:=0;  //default
mb_Output_Registers[85]:=0;  //default
mb_Output_Registers[86]:=0;  //default
mb_Output_Registers[87]:=0;  //default
mb_Output_Registers[88]:=0;  //default
mb_Output_Registers[89]:=0;  //default
mb_Output_Registers[90]:=0;  //default
mb_Output_Registers[91]:=0;  //default
mb_Output_Registers[92]:=0;  //default
mb_Output_Registers[93]:=0;  //default
mb_Output_Registers[94]:=0;  //default
mb_Output_Registers[95]:=0;  //default
mb_Output_Registers[96]:=0;  //default
mb_Output_Registers[97]:=0;  //default
mb_Output_Registers[98]:=0;  //default
mb_Output_Registers[99]:=0;  //default
mb_Output_Registers[100]:=0;  //default
mb_Output_Registers[101]:=0;  //default
mb_Output_Registers[102]:=0;  //default
mb_Output_Registers[103]:=0;  //default
mb_Output_Registers[104]:=0;  //default
mb_Output_Registers[105]:=0;  //default
mb_Output_Registers[106]:=0;  //default
mb_Output_Registers[107]:=0;  //default
mb_Output_Registers[108]:=0;  //default
mb_Output_Registers[109]:=0;  //default
mb_Output_Registers[110]:=0;  //default
mb_Output_Registers[111]:=0;  //default
mb_Output_Registers[112]:=0;  //default
mb_Output_Registers[113]:=0;  //default
mb_Output_Registers[114]:=0;  //default
mb_Output_Registers[115]:=0;  //default
mb_Output_Registers[116]:=0;  //default
mb_Output_Registers[117]:=0;  //default
mb_Output_Registers[118]:=0;  //default
mb_Output_Registers[119]:=0;  //default
mb_Output_Registers[120]:=0;  //default
mb_Output_Registers[121]:=0;  //default
mb_Output_Registers[122]:=0;  //default
mb_Output_Registers[123]:=0;  //default
mb_Output_Registers[124]:=0;  //default
mb_Output_Registers[125]:=0;  //default
mb_Output_Registers[126]:=0;  //default
mb_Output_Registers[127]:=0;  //default
mb_Output_Registers[128]:=0;  //default
mb_Output_Registers[129]:=0;  //default
mb_Output_Registers[130]:=0;  //default
mb_Output_Registers[131]:=0;  //default
mb_Output_Registers[132]:=0;  //default
mb_Output_Registers[133]:=0;  //default
mb_Output_Registers[134]:=0;  //default
mb_Output_Registers[135]:=0;  //default
mb_Output_Registers[136]:=0;  //default
mb_Output_Registers[137]:=0;  //default
mb_Output_Registers[138]:=0;  //default
mb_Output_Registers[139]:=0;  //default
mb_Output_Registers[140]:=0;  //default
mb_Output_Registers[141]:=0;  //default
mb_Output_Registers[142]:=0;  //default
mb_Output_Registers[143]:=0;  //default
mb_Output_Registers[144]:=0;  //default
mb_Output_Registers[145]:=0;  //default
mb_Output_Registers[146]:=0;  //default
mb_Output_Registers[147]:=0;  //default
mb_Output_Registers[148]:=0;  //default
mb_Output_Registers[149]:=0;  //default
mb_Output_Registers[150]:=0;  //default
mb_Output_Registers[151]:=0;  //default
mb_Output_Registers[152]:=0;  //default
mb_Output_Registers[153]:=0;  //default
mb_Output_Registers[154]:=0;  //default
mb_Output_Registers[155]:=0;  //default
mb_Output_Registers[156]:=0;  //default
mb_Output_Registers[157]:=0;  //default
mb_Output_Registers[158]:=0;  //default
mb_Output_Registers[159]:=0;  //default
mb_Output_Registers[160]:=0;  //default
mb_Output_Registers[161]:=0;  //default
mb_Output_Registers[162]:=0;  //default
mb_Output_Registers[163]:=0;  //default
mb_Output_Registers[164]:=0;  //default
mb_Output_Registers[165]:=0;  //default
mb_Output_Registers[166]:=0;  //default
mb_Output_Registers[167]:=0;  //default
mb_Output_Registers[168]:=0;  //default
mb_Output_Registers[169]:=0;  //default
mb_Output_Registers[170]:=0;  //default
mb_Output_Registers[171]:=0;  //default
mb_Output_Registers[172]:=0;  //default
mb_Output_Registers[173]:=0;  //default
mb_Output_Registers[174]:=0;  //default
mb_Output_Registers[175]:=0;  //default
mb_Output_Registers[176]:=0;  //default
mb_Output_Registers[177]:=0;  //default
mb_Output_Registers[178]:=0;  //default
mb_Output_Registers[179]:=0;  //default
mb_Output_Registers[180]:=0;  //default
mb_Output_Registers[181]:=0;  //default
mb_Output_Registers[182]:=0;  //default
mb_Output_Registers[183]:=0;  //default
mb_Output_Registers[184]:=0;  //default
mb_Output_Registers[185]:=0;  //default
mb_Output_Registers[186]:=0;  //default
mb_Output_Registers[187]:=0;  //default
mb_Output_Registers[188]:=0;  //default
mb_Output_Registers[189]:=0;  //default
mb_Output_Registers[190]:=0;  //default
mb_Output_Registers[191]:=0;  //default
mb_Output_Registers[192]:=0;  //default
mb_Output_Registers[193]:=0;  //default
mb_Output_Registers[194]:=0;  //default
mb_Output_Registers[195]:=0;  //default
mb_Output_Registers[196]:=0;  //default
mb_Output_Registers[197]:=0;  //default
mb_Output_Registers[198]:=0;  //default
mb_Output_Registers[199]:=0;  //default
mb_Output_Registers[200]:=0;  //default
mb_Output_Registers[201]:=0;  //default
mb_Output_Registers[202]:=0;  //default
mb_Output_Registers[203]:=0;  //default
mb_Output_Registers[204]:=0;  //default
mb_Output_Registers[205]:=0;  //default
mb_Output_Registers[206]:=0;  //default
mb_Output_Registers[207]:=0;  //default
mb_Output_Registers[208]:=0;  //default
mb_Output_Registers[209]:=0;  //default
mb_Output_Registers[210]:=0;  //default
mb_Output_Registers[211]:=0;  //default
mb_Output_Registers[212]:=0;  //default
mb_Output_Registers[213]:=0;  //default
mb_Output_Registers[214]:=0;  //default
mb_Output_Registers[215]:=0;  //default
mb_Output_Registers[216]:=0;  //default
mb_Output_Registers[217]:=0;  //default
mb_Output_Registers[218]:=0;  //default
mb_Output_Registers[219]:=0;  //default
mb_Output_Registers[220]:=0;  //default
mb_Output_Registers[221]:=0;  //default
mb_Output_Registers[222]:=0;  //default
mb_Output_Registers[223]:=0;  //default
mb_Output_Registers[224]:=0;  //default
mb_Output_Registers[225]:=0;  //default
mb_Output_Registers[226]:=0;  //default
mb_Output_Registers[227]:=0;  //default
mb_Output_Registers[228]:=0;  //default
mb_Output_Registers[229]:=0;  //default
mb_Output_Registers[230]:=0;  //default
mb_Output_Registers[231]:=0;  //default
mb_Output_Registers[232]:=0;  //default
mb_Output_Registers[233]:=0;  //default
mb_Output_Registers[234]:=0;  //default
mb_Output_Registers[235]:=0;  //default
mb_Output_Registers[236]:=0;  //default
mb_Output_Registers[237]:=0;  //default
mb_Output_Registers[238]:=0;  //default
mb_Output_Registers[239]:=0;  //default
mb_Output_Registers[240]:=0;  //default
mb_Output_Registers[241]:=0;  //default
mb_Output_Registers[242]:=0;  //default
mb_Output_Registers[243]:=0;  //default
mb_Output_Registers[244]:=0;  //default
mb_Output_Registers[245]:=0;  //default
mb_Output_Registers[246]:=0;  //default
mb_Output_Registers[247]:=0;  //default
mb_Output_Registers[248]:=0;  //default
mb_Output_Registers[249]:=0;  //default
mb_Output_Registers[250]:=0;  //default
mb_Output_Registers[251]:=0;  //default
mb_Output_Registers[252]:=0;  //default
mb_Output_Registers[253]:=0;  //default
mb_Output_Registers[254]:=0;  //default
mb_Output_Registers[255]:=0;  //default

END_PROGRAM

// ---- POUs/Modbus/p_ModbusTx_PLCMemory.TcPOU
PROGRAM p_ModbusTx_PLCMemory
VAR
END_VAR

(*mb_PLC_Memory[0]-[99] PLC aiFloat inputs *)


MEMCPY(destAddr:=ADR(mb_PLC_Memory[10]), srcAddr:=ADR(vgPBT_GCC_02.rPRESS), n:=SIZEOF(vgPBT_GCC_02.rPRESS));  //VG pressure readbacks
MEMCPY(destAddr:=ADR(mb_PLC_Memory[12]), srcAddr:=ADR(vgPBT_GPI_02.rPRESS), n:=SIZEOF(vgPBT_GPI_02.rPRESS));  //VG pressure readbacks

MEMCPY(destAddr:=ADR(mb_PLC_Memory[14]), srcAddr:=ADR(vgPBT_GCC_04.rPRESS), n:=SIZEOF(vgPBT_GCC_04.rPRESS));  //VG pressure readbacks
MEMCPY(destAddr:=ADR(mb_PLC_Memory[16]), srcAddr:=ADR(vgPBT_GPI_04.rPRESS), n:=SIZEOF(vgPBT_GPI_04.rPRESS));  //VG pressure readbacks

MEMCPY(destAddr:=ADR(mb_PLC_Memory[18]), srcAddr:=ADR(vgPBT_GCC_06.rPRESS), n:=SIZEOF(vgPBT_GCC_06.rPRESS));  //VG pressure readbacks
MEMCPY(destAddr:=ADR(mb_PLC_Memory[20]), srcAddr:=ADR(vgPBT_GPI_06.rPRESS), n:=SIZEOF(vgPBT_GPI_06.rPRESS));  //VG pressure readbacks

MEMCPY(destAddr:=ADR(mb_PLC_Memory[22]), srcAddr:=ADR(vgPBT_GCC_07.rPRESS), n:=SIZEOF(vgPBT_GCC_07.rPRESS));  //VG pressure readbacks
MEMCPY(destAddr:=ADR(mb_PLC_Memory[24]), srcAddr:=ADR(vgPBT_GPI_07.rPRESS), n:=SIZEOF(vgPBT_GPI_07.rPRESS));  //VG pressure readbacks

MEMCPY(destAddr:=ADR(mb_PLC_Memory[26]), srcAddr:=ADR(vgPBT_GCC_09.rPRESS), n:=SIZEOF(vgPBT_GCC_09.rPRESS));  //VG pressure readbacks
MEMCPY(destAddr:=ADR(mb_PLC_Memory[28]), srcAddr:=ADR(vgPBT_GPI_09.rPRESS), n:=SIZEOF(vgPBT_GPI_09.rPRESS));  //VG pressure readbacks

END_PROGRAM

// ---- POUs/Modbus/p_XLegacyPLCModbus.TcPOU
PROGRAM p_XLegacyPLCModbus
VAR
	fbHFX_PLCInputCoilsRx	:	FB_MBReadInputs;
	
	i_xHFX_PLC_CnBits	:	ARRAY [0..20] OF BYTE;
	
	ftResetHFX	: F_TRIG; 
	tonRetryHFX : TON;
END_VAR


(* Modbus Info for Koyo
Modbus Addresses for
Koyo DL05/06/240/250/260/430/440/450 PLCs
PLC Memory Type		| Modbus start address Decimal (octal) | Function codes
Inputs (X)			  2048 (04000)							2
Special Relays (SP)	  3072 (06000)							2
Outputs (Y)			  2048 (04000)							1, 5, 15
Control Relays (C)	  3072 (06000)							1, 5, 15
Timer Contacts (T)	  6144 (014000)							1, 5, 15
Counter Contacts (CT) 6400 (014400)							1, 5, 15
Stage Status Bits (S) 6144 (012000)							1, 5, 15
*)


(* HFX code *)
// Retry after some time
tonRetryHFX.IN := NOT fbHFX_PLCInputCoilsRx.bBusy;
tonRetryHFX.PT := T#10S;
tonRetryHFX();

ftResetHFX(CLK:=fbHFX_PLCInputCoilsRx.bBusy);
//ftResetHFX();

fbHFX_PLCInputCoilsRx.bExecute := ftResetHFX.Q OR tonRetryHFX.Q;

fbHFX_PLCInputCoilsRx(sIPAddr:='172.21.88.95', nTCPPort:=502, nQuantity:=32, nMBAddr:=8#6000, cbLength:=SIZEOF(i_xHFX_PLC_CnBits),  pDestAddr:=ADR(i_xHFX_PLC_CnBits), tTimeout:=T#5S);

IF fbHFX_PLCInputCoilsRx.bError THEN
	//run some error code for modbus
	//if there's a modbus error, set all incoming bits to zero
	// HFX PLC Relay coil C[3] is used for PBT downstream VacOK
	i_xHFX_PLC_CnBits[0].0 := 0;
	i_xHFX_PLC_CnBits[0].1 := 0;
	i_xHFX_PLC_CnBits[0].2 := 0;
	i_xHFX_PLC_CnBits[0].3 := 0;
	i_xHFX_PLC_CnBits[0].4 := 0;
	i_xHFX_PLC_CnBits[1].0 := 0;
	i_xHFX_PLC_CnBits[1].1 := 0;
	i_xHFX_PLC_CnBits[1].2 := 0;
	g_ixDSVacOK := FALSE;
	g_xNoHFXPLCResponse:= TRUE;
	
	
ELSIF Not ftResetHFX.Q AND fbHFX_PLCInputCoilsRx.cbRead > 0 THEN
	g_xNoHFXPLCResponse:= FALSE;
	g_ixDSVacOK := i_xHFX_PLC_CnBits[0].2;
	fbHFX_PLCInputCoilsRx.bExecute :=False;
ELSIF ftResetHFX.Q AND fbHFX_PLCInputCoilsRx.cbRead = 0 THEN
	//more error code cause we didn't manage to read anything
	//g_ixDSVacOK := FALSE;
	//g_xNoHFXPLCResponse:= TRUE;
			
END_IF

END_PROGRAM
